//点样轴6X伺服控制
FB_SERVOAXIS_3(
	AXIS:= 点样轴6X ,                    //轴名称
	xEnable:=急停  ,                         //轴使能
	xStartupMotionAllowed:= FALSE, // startup axis ownership
	xHome:= 点样轴6XDATE.xHome,          //轴回零命令
	xJogPos:=点样轴6XDATE.xJogPos  ,     //轴正转命令
	xJogNeg:=点样轴6XDATE.xJogNeg  ,     //轴反转命令
	xStop:= 点样轴6XDATE.xStop ,         //轴停止命令
	xMoveAbs:= 点样轴6XDATE.xMoveAbs ,   //轴绝对定位命令
	xMoveRel:= 点样轴6XDATE.xMoveRel,    //轴相对定位命令
	XReset:= 点样轴6XDATE.XReset OR 复位 OR bSysReset,       //轴复位
	fAbsTarget:= 点样轴6XDATE.fAbsTarget ,  //轴绝对定位距离
	fRelTarget:=点样轴6XDATE.fRelTarget  ,  //轴相对移动距离
	fVelocity:= 点样轴6XDATE.fVelocity ,    //轴定位速度
	fAcc:=3500.0 ,              //轴加速度
	fDec:= 3500.0,              //轴减速度
	fJogVel:= 50.0 ,        //轴JOG速度
	bEnabled=> 点样轴6XDATE.bEnabled ,      //轴使能完成
	bHomed=> 回零完成6X ,          //轴回原点完成
	bBusy=> 点样轴6XDATE.bBusy ,            //轴运行中
	fActPos=>点样轴6XDATE.fActPos  ,        //轴当前位置
	fActVel=>点样轴6XDATE.fActVel  ,        //轴当前速度
	bAbMoveDone=>点样轴6XDATE.bAbMoveDone ,  //轴绝对定位完成
	bReMoveDone =>点样轴6XDATE.bReMoveDone ,);    //轴相对定位完成 
// startup alarm visibility axis 3
点样轴6XDATE.bError := FB_SERVOAXIS_3.bError AND NOT PLC_Startup_AlarmInhibit;
IF PLC_Startup_AlarmInhibit THEN
	点样轴6XDATE.iErrorCode := 0;
ELSE
	点样轴6XDATE.iErrorCode := FB_SERVOAXIS_3.iErrorCode;
END_IF
IF 回零完成6X THEN
	点样轴6XDATE.xHome := FALSE;
	点样轴6XDATE.bHomed := TRUE;
END_IF

//点样轴7Y伺服控制
FB_SERVOAXIS_4(
	AXIS:= 点样轴7Y ,                    //轴名称
	xEnable:=急停  ,                         //轴使能
	xStartupMotionAllowed:= FALSE, // startup axis ownership
	xHome:= 点样轴7YDATE.xHome,          //轴回零命令
	xJogPos:=点样轴7YDATE.xJogPos  ,     //轴正转命令
	xJogNeg:=点样轴7YDATE.xJogNeg  ,     //轴反转命令
	xStop:= 点样轴7YDATE.xStop ,         //轴停止命令
	xMoveAbs:= 点样轴7YDATE.xMoveAbs ,   //轴绝对定位命令
	xMoveRel:= 点样轴7YDATE.xMoveRel,    //轴相对定位命令
	XReset:= 点样轴7YDATE.XReset OR 复位 OR bSysReset,       //轴复位
	fAbsTarget:= 点样轴7YDATE.fAbsTarget ,  //轴绝对定位距离
	fRelTarget:=点样轴7YDATE.fRelTarget  ,  //轴相对移动距离
	fVelocity:= 点样轴7YDATE.fVelocity ,    //轴定位速度
	fAcc:=500.0 ,              //轴加速度
	fDec:= 500.0 ,              //轴减速度
	fJogVel:= 50.0 ,        //轴JOG速度
	bEnabled=> 点样轴7YDATE.bEnabled ,      //轴使能完成
	bHomed=>  回零完成7Y,          //轴回原点完成
	bBusy=> 点样轴7YDATE.bBusy ,            //轴运行中
	fActPos=>点样轴7YDATE.fActPos  ,        //轴当前位置
	fActVel=>点样轴7YDATE.fActVel  ,        //轴当前速度
	bAbMoveDone=>点样轴7YDATE.bAbMoveDone ,  //轴绝对定位完成
	bReMoveDone =>点样轴7YDATE.bReMoveDone ,);    //轴相对定位完成 
// startup alarm visibility axis 4
点样轴7YDATE.bError := FB_SERVOAXIS_4.bError AND NOT PLC_Startup_AlarmInhibit;
IF PLC_Startup_AlarmInhibit THEN
	点样轴7YDATE.iErrorCode := 0;
ELSE
	点样轴7YDATE.iErrorCode := FB_SERVOAXIS_4.iErrorCode;
END_IF
IF 回零完成7Y THEN
	点样轴7YDATE.xHome := FALSE;
	点样轴7YDATE.bHomed := TRUE;
END_IF

//拍照轴8Y伺服控制
FB_SERVOAXIS_5(
	AXIS:= 拍照轴8Y ,                    //轴名称
	xEnable:=急停  ,                         //轴使能
	xStartupMotionAllowed:= FALSE, // startup axis ownership
	xHome:= 拍照轴8YDATE.xHome,          //轴回零命令
	xJogPos:=拍照轴8YDATE.xJogPos  ,     //轴正转命令
	xJogNeg:=拍照轴8YDATE.xJogNeg  ,     //轴反转命令
	xStop:= 拍照轴8YDATE.xStop ,         //轴停止命令
	xMoveAbs:= 拍照轴8YDATE.xMoveAbs AND  刮板拍照遮光气缸上位 AND 刮板轴10ZDATE.fActPos<6 ,   //轴绝对定位命令
	xMoveRel:= 拍照轴8YDATE.xMoveRel,    //轴相对定位命令
	XReset:= 拍照轴8YDATE.XReset OR 复位 OR bSysReset,       //轴复位
	fAbsTarget:= 拍照轴8YDATE.fAbsTarget ,  //轴绝对定位距离
	fRelTarget:=拍照轴8YDATE.fRelTarget  ,  //轴相对移动距离
	fVelocity:= 拍照轴8YDATE.fVelocity ,    //轴定位速度
	fAcc:=500.0 ,              //轴加速度
	fDec:= 500.0 ,              //轴减速度
	fJogVel:= 50.0 ,        //轴JOG速度
	bEnabled=> 拍照轴8YDATE.bEnabled ,      //轴使能完成
	bHomed=> 回零完成8Y ,          //轴回原点完成
	bBusy=> 拍照轴8YDATE.bBusy ,            //轴运行中
	fActPos=>拍照轴8YDATE.fActPos  ,        //轴当前位置
	fActVel=>拍照轴8YDATE.fActVel  ,        //轴当前速度
	bAbMoveDone=>拍照轴8YDATE.bAbMoveDone ,  //轴绝对定位完成
	bReMoveDone =>拍照轴8YDATE.bReMoveDone ,);    //轴相对定位完成 
// startup alarm visibility axis 5
拍照轴8YDATE.bError := FB_SERVOAXIS_5.bError AND NOT PLC_Startup_AlarmInhibit;
IF PLC_Startup_AlarmInhibit THEN
	拍照轴8YDATE.iErrorCode := 0;
ELSE
	拍照轴8YDATE.iErrorCode := FB_SERVOAXIS_5.iErrorCode;
END_IF
	IF 回零完成8Y THEN
	拍照轴8YDATE.xHome := FALSE;
	拍照轴8YDATE.bHomed := TRUE;
END_IF

//刮板轴9X伺服控制
FB_SERVOAXIS_6(
	AXIS:= 刮板轴9X ,                    //轴名称
	xEnable:=急停  ,                         //轴使能
	xStartupMotionAllowed:= FALSE, // startup axis ownership
	xHome:= 刮板轴9XDATE.xHome,          //轴回零命令
	xJogPos:=刮板轴9XDATE.xJogPos  ,     //轴正转命令
	xJogNeg:=刮板轴9XDATE.xJogNeg  ,     //轴反转命令
	xStop:= 刮板轴9XDATE.xStop ,         //轴停止命令
	xMoveAbs:= 刮板轴9XDATE.xMoveAbs AND  刮板轴10ZDATE.fActPos<6,   //轴绝对定位命令
	xMoveRel:= 刮板轴9XDATE.xMoveRel,    //轴相对定位命令
	XReset:= 刮板轴9XDATE.XReset OR 复位 OR bSysReset,       //轴复位
	fAbsTarget:= 刮板轴9XDATE.fAbsTarget  ,  //轴绝对定位距离
	fRelTarget:=刮板轴9XDATE.fRelTarget  ,  //轴相对移动距离
	fVelocity:= 刮板轴9XDATE.fVelocity ,    //轴定位速度
	fAcc:=500.0 ,              //轴加速度
	fDec:= 500.0 ,              //轴减速度
	fJogVel:= 50.0 ,        //轴JOG速度
	bEnabled=> 刮板轴9XDATE.bEnabled ,      //轴使能完成
	bHomed=>  回零完成9X,          //轴回原点完成
	bBusy=> 刮板轴9XDATE.bBusy ,            //轴运行中
	fActPos=>刮板轴9XDATE.fActPos  ,        //轴当前位置
	fActVel=>刮板轴9XDATE.fActVel  ,        //轴当前速度
	bAbMoveDone=>刮板轴9XDATE.bAbMoveDone ,  //轴绝对定位完成
	bReMoveDone =>刮板轴9XDATE.bReMoveDone ,);    //轴相对定位完成 
// startup alarm visibility axis 6
刮板轴9XDATE.bError := FB_SERVOAXIS_6.bError AND NOT PLC_Startup_AlarmInhibit;
IF PLC_Startup_AlarmInhibit THEN
	刮板轴9XDATE.iErrorCode := 0;
ELSE
	刮板轴9XDATE.iErrorCode := FB_SERVOAXIS_6.iErrorCode;
END_IF
IF 回零完成9X THEN
	刮板轴9XDATE.xHome := FALSE;
	刮板轴9XDATE.bHomed := TRUE;
END_IF

//刮板轴10Z伺服控制
FB_SERVOAXIS_7(
	AXIS:= 刮板轴10Z ,                    //轴名称
	xEnable:=急停  ,                         //轴使能
	xStartupMotionAllowed:= FALSE, // startup axis ownership
	xHome:= 刮板轴10ZDATE.xHome,          //轴回零命令
	xJogPos:=刮板轴10ZDATE.xJogPos  ,     //轴正转命令
	xJogNeg:=刮板轴10ZDATE.xJogNeg  ,     //轴反转命令
	xStop:= 刮板轴10ZDATE.xStop ,         //轴停止命令
	xMoveAbs:= 刮板轴10ZDATE.xMoveAbs ,   //轴绝对定位命令
	xMoveRel:= 刮板轴10ZDATE.xMoveRel,    //轴相对定位命令
	XReset:= 刮板轴10ZDATE.XReset OR 复位 OR bSysReset,       //轴复位
	fAbsTarget:= 刮板轴10ZDATE.fAbsTarget ,  //轴绝对定位距离
	fRelTarget:=刮板轴10ZDATE.fRelTarget  ,  //轴相对移动距离
	fVelocity:= 刮板轴10ZDATE.fVelocity ,    //轴定位速度
	fAcc:=500.0  ,              //轴加速度
	fDec:= 500.0 ,              //轴减速度
	fJogVel:= 50.0 ,        //轴JOG速度
	bEnabled=> 刮板轴10ZDATE.bEnabled ,      //轴使能完成
	bHomed=> 回零完成10Z ,          //轴回原点完成
	bBusy=> 刮板轴10ZDATE.bBusy ,            //轴运行中
	fActPos=>刮板轴10ZDATE.fActPos  ,        //轴当前位置
	fActVel=>刮板轴10ZDATE.fActVel  ,        //轴当前速度
	bAbMoveDone=>刮板轴10ZDATE.bAbMoveDone ,  //轴绝对定位完成
	bReMoveDone =>刮板轴10ZDATE.bReMoveDone ,);    //轴相对定位完成 
// startup alarm visibility axis 7
刮板轴10ZDATE.bError := FB_SERVOAXIS_7.bError AND NOT PLC_Startup_AlarmInhibit;
IF PLC_Startup_AlarmInhibit THEN
	刮板轴10ZDATE.iErrorCode := 0;
ELSE
	刮板轴10ZDATE.iErrorCode := FB_SERVOAXIS_7.iErrorCode;
END_IF
IF 回零完成10Z THEN
	刮板轴10ZDATE.xHome := FALSE;
	刮板轴10ZDATE.bHomed := TRUE;
END_IF	
	
//地轨轴11Y伺服控制
FB_SERVOAXIS_8(
	AXIS:= 地轨轴11Y ,                    //轴名称
	xEnable:=急停  ,                         //轴使能
	xStartupMotionAllowed:= FALSE, // startup axis ownership
	xHome:= 地轨轴11YDATE.xHome,          //轴回零命令
	xJogPos:=地轨轴11YDATE.xJogPos  ,     //轴正转命令
	xJogNeg:=地轨轴11YDATE.xJogNeg  ,     //轴反转命令
	xStop:= 地轨轴11YDATE.xStop ,         //轴停止命令
	xMoveAbs:= 地轨轴11YDATE.xMoveAbs  ,   //轴绝对定位命令
	xMoveRel:= 地轨轴11YDATE.xMoveRel,    //轴相对定位命令
	XReset:= 地轨轴11YDATE.XReset OR 复位 OR bSysReset,       //轴复位
	fAbsTarget:= 地轨轴11YDATE.fAbsTarget ,  //轴绝对定位距离
	fRelTarget:=地轨轴11YDATE.fRelTarget  ,  //轴相对移动距离
	fVelocity:= 地轨轴11YDATE.fVelocity ,    //轴定位速度
	fAcc:=500.0 ,              //轴加速度
	fDec:= 500.0 ,              //轴减速度
	fJogVel:= 50.0 ,        //轴JOG速度
	bEnabled=> 地轨轴11YDATE.bEnabled ,      //轴使能完成
	bHomed=>  回零完成11Y,          //轴回原点完成
	bBusy=> 地轨轴11YDATE.bBusy ,            //轴运行中
	fActPos=>地轨轴11YDATE.fActPos  ,        //轴当前位置
	fActVel=>地轨轴11YDATE.fActVel  ,        //轴当前速度
	bAbMoveDone=>地轨轴11YDATE.bAbMoveDone ,  //轴绝对定位完成
	bReMoveDone =>地轨轴11YDATE.bReMoveDone ,);    //轴相对定位完成 
// startup alarm visibility axis 8
地轨轴11YDATE.bError := FB_SERVOAXIS_8.bError AND NOT PLC_Startup_AlarmInhibit;
IF PLC_Startup_AlarmInhibit THEN
	地轨轴11YDATE.iErrorCode := 0;
ELSE
	地轨轴11YDATE.iErrorCode := FB_SERVOAXIS_8.iErrorCode;
END_IF
IF 回零完成11Y THEN
	地轨轴11YDATE.xHome := FALSE;
	地轨轴11YDATE.bHomed := TRUE;
END_IF

//上样轴4X轴伺服控制
FB_SERVOAXIS_9(
	AXIS:= 上样轴4X轴 ,                    //轴名称
	xEnable:= 急停 AND NOT (Sampling_Servo_FreeMove AND (上样轴5Z轴DATE.fActPos < 3)) ,   //轴使能(去使能手推: 仅5Z抬起<3时放开4X)
	xStartupMotionAllowed:= ((PLC_Startup_State=50) OR (PLC_Startup_State=51)), // startup axis ownership
	xHome:= 上样轴4X轴DATE.xHome,          //轴回零命令
	xJogPos:=上样轴4X轴DATE.xJogPos  ,     //轴正转命令
	xJogNeg:=上样轴4X轴DATE.xJogNeg  ,     //轴反转命令
	xStop:= 上样轴4X轴DATE.xStop ,         //轴停止命令
	xMoveAbs:= 上样轴4X轴DATE.xMoveAbs AND  上样轴5Z轴DATE.fActPos<3 ,   //轴绝对定位命令
	xMoveRel:= 上样轴4X轴DATE.xMoveRel AND  上样轴5Z轴DATE.fActPos<3,    //轴相对定位命令
	XReset:= 上样轴4X轴DATE.XReset OR 复位 OR bSysReset,       //轴复位
	fAbsTarget:= 上样轴4X轴DATE.fAbsTarget ,  //轴绝对定位距离
	fRelTarget:=上样轴4X轴DATE.fRelTarget  ,  //轴相对移动距离
	fVelocity:= 上样轴4X轴DATE.fVelocity ,    //轴定位速度
	fAcc:=200.0 ,              //轴加速度
	fDec:= 200.0 ,              //轴减速度
	fJogVel:= 5.0,        //轴JOG速度
	bEnabled=> 上样轴4X轴DATE.bEnabled ,      //轴使能完成
	bHomed=>  回零完成4X,          //轴回原点完成
	bBusy=> 上样轴4X轴DATE.bBusy ,            //轴运行中
	fActPos=>上样轴4X轴DATE.fActPos  ,        //轴当前位置
	fActVel=>上样轴4X轴DATE.fActVel  ,        //轴当前速度
	bAbMoveDone=>上样轴4X轴DATE.bAbMoveDone ,  //轴绝对定位完成
	bReMoveDone =>上样轴4X轴DATE.bReMoveDone ,);    //轴相对定位完成 
// startup alarm visibility axis 9
上样轴4X轴DATE.bError := FB_SERVOAXIS_9.bError AND NOT PLC_Startup_AlarmInhibit;
IF PLC_Startup_AlarmInhibit THEN
	上样轴4X轴DATE.iErrorCode := 0;
ELSE
	上样轴4X轴DATE.iErrorCode := FB_SERVOAXIS_9.iErrorCode;
END_IF
IF 回零完成4X THEN
	上样轴4X轴DATE.xHome := FALSE;
	上样轴4X轴DATE.bHomed := TRUE;
END_IF
	%QB2216:= 27;             //回零模式27
IF NOT 急停 THEN
	上样轴4X轴DATE.bHomed := FALSE;
END_IF

//上样轴5Z轴伺服控制
FB_SERVOAXIS_10(
	AXIS:= 上样轴5Z轴 ,                    //轴名称
	xEnable:=急停  ,                         //轴使能
	xStartupMotionAllowed:= ((PLC_Startup_State=40) OR (PLC_Startup_State=41)), // startup axis ownership
	xHome:= 上样轴5Z轴DATE.xHome,          //轴回零命令
	xJogPos:=上样轴5Z轴DATE.xJogPos  ,     //轴正转命令
	xJogNeg:=上样轴5Z轴DATE.xJogNeg  ,     //轴反转命令
	xStop:= 上样轴5Z轴DATE.xStop ,         //轴停止命令
	xMoveAbs:= 上样轴5Z轴DATE.xMoveAbs ,   //轴绝对定位命令
	xMoveRel:= 上样轴5Z轴DATE.xMoveRel,    //轴相对定位命令
	XReset:= 上样轴5Z轴DATE.XReset OR 复位 OR bSysReset ,       //轴复位
	fAbsTarget:= 上样轴5Z轴DATE.fAbsTarget ,  //轴绝对定位距离
	fRelTarget:=上样轴5Z轴DATE.fRelTarget  ,  //轴相对移动距离
	fVelocity:= 上样轴5Z轴DATE.fVelocity ,    //轴定位速度
	fAcc:=300.0  ,              //轴加速度
	fDec:= 300.0 ,              //轴减速度
	fJogVel:= 20.0 ,        //轴JOG速度
	bEnabled=> 上样轴5Z轴DATE.bEnabled ,      //轴使能完成
	bHomed=> 回零完成5Z ,          //轴回原点完成
	bBusy=> 上样轴5Z轴DATE.bBusy ,            //轴运行中
	fActPos=>上样轴5Z轴DATE.fActPos  ,        //轴当前位置
	fActVel=>上样轴5Z轴DATE.fActVel  ,        //轴当前速度
	bAbMoveDone=>上样轴5Z轴DATE.bAbMoveDone ,   //轴绝对定位完成
	bReMoveDone =>上样轴5Z轴DATE.bReMoveDone , );   //轴相对定位完成 
// startup alarm visibility axis 10
上样轴5Z轴DATE.bError := FB_SERVOAXIS_10.bError AND NOT PLC_Startup_AlarmInhibit;
IF PLC_Startup_AlarmInhibit THEN
	上样轴5Z轴DATE.iErrorCode := 0;
ELSE
	上样轴5Z轴DATE.iErrorCode := FB_SERVOAXIS_10.iErrorCode;
END_IF
IF 回零完成5Z THEN
	上样轴5Z轴DATE.xHome := FALSE;
	上样轴5Z轴DATE.bHomed := TRUE;
END_IF
	%QB2228:= 27;                 //回零模式27
IF NOT 急停 THEN
	上样轴5Z轴DATE.bHomed := FALSE;
END_IF

//上样4X 与 打样3Y 实际使能镜像 -> 供上位机标定页显示真状态 (去使能手推时为 FALSE)
Sampling_Servo_Enabled := 上样轴4X轴DATE.bEnabled AND 打样瓶上料轴3YDATE.bEnabled;
END_ACTION

ACTION 位置示教:

//打样瓶上料轴3Y位置示教
FB_Teach_1(HMI_Servo:=HMI_打样瓶上料轴3Y , 
			Servo:=打样瓶上料轴3YDATE );
//点样轴6X位置示教
FB_Teach_2(HMI_Servo:=HMI_点样轴6X , 
			Servo:=点样轴6XDATE );
//点样轴7Y位置示教
FB_Teach_3(HMI_Servo:=HMI_点样轴7Y , 
			Servo:=点样轴7YDATE );			
//地轨轴11Y位置示教
FB_Teach_4(HMI_Servo:=HMI_地轨轴11Y , 
			Servo:=地轨轴11YDATE );			
//上样轴4X轴位置示教
FB_Teach_5(HMI_Servo:=HMI_上样轴4X轴 , 
			Servo:=上样轴4X轴DATE );			
//上样轴5Z轴位置示教
FB_Teach_6(HMI_Servo:=HMI_上样轴5Z轴 , 
			Servo:=上样轴5Z轴DATE );
END_ACTION

END_PROGRAM

// Device/Application/40_Man/initialization
PROGRAM initialization
VAR
	nTeachClear : INT;

END_VAR

玻璃上料轴1ZDATE.xHome := FALSE; 玻璃上料轴1ZDATE.xJogPos := FALSE; 玻璃上料轴1ZDATE.xJogNeg := FALSE;
玻璃上料轴1ZDATE.xMoveAbs := FALSE; 玻璃上料轴1ZDATE.xMoveRel := FALSE; 玻璃上料轴1ZDATE.xStop := FALSE; 玻璃上料轴1ZDATE.XReset := FALSE;
玻璃上料轴1ZDATE.bBusy := FALSE; 玻璃上料轴1ZDATE.bError := FALSE; 玻璃上料轴1ZDATE.iErrorCode := 0;
玻璃上料轴1ZDATE.bAbMoveDone := FALSE; 玻璃上料轴1ZDATE.bReMoveDone := FALSE;
玻璃上料轴2ZDATE.xHome := FALSE; 玻璃上料轴2ZDATE.xJogPos := FALSE; 玻璃上料轴2ZDATE.xJogNeg := FALSE;
玻璃上料轴2ZDATE.xMoveAbs := FALSE; 玻璃上料轴2ZDATE.xMoveRel := FALSE; 玻璃上料轴2ZDATE.xStop := FALSE; 玻璃上料轴2ZDATE.XReset := FALSE;
玻璃上料轴2ZDATE.bBusy := FALSE; 玻璃上料轴2ZDATE.bError := FALSE; 玻璃上料轴2ZDATE.iErrorCode := 0;
玻璃上料轴2ZDATE.bAbMoveDone := FALSE; 玻璃上料轴2ZDATE.bReMoveDone := FALSE;
打样瓶上料轴3YDATE.xHome := FALSE; 打样瓶上料轴3YDATE.xJogPos := FALSE; 打样瓶上料轴3YDATE.xJogNeg := FALSE;
打样瓶上料轴3YDATE.xMoveAbs := FALSE; 打样瓶上料轴3YDATE.xMoveRel := FALSE; 打样瓶上料轴3YDATE.xStop := FALSE; 打样瓶上料轴3YDATE.XReset := FALSE;
打样瓶上料轴3YDATE.bBusy := FALSE; 打样瓶上料轴3YDATE.bError := FALSE; 打样瓶上料轴3YDATE.iErrorCode := 0;
打样瓶上料轴3YDATE.bAbMoveDone := FALSE; 打样瓶上料轴3YDATE.bReMoveDone := FALSE;
点样轴6XDATE.xHome := FALSE; 点样轴6XDATE.xJogPos := FALSE; 点样轴6XDATE.xJogNeg := FALSE;
点样轴6XDATE.xMoveAbs := FALSE; 点样轴6XDATE.xMoveRel := FALSE; 点样轴6XDATE.xStop := FALSE; 点样轴6XDATE.XReset := FALSE;
点样轴6XDATE.bBusy := FALSE; 点样轴6XDATE.bError := FALSE; 点样轴6XDATE.iErrorCode := 0;
点样轴6XDATE.bAbMoveDone := FALSE; 点样轴6XDATE.bReMoveDone := FALSE;
点样轴7YDATE.xHome := FALSE; 点样轴7YDATE.xJogPos := FALSE; 点样轴7YDATE.xJogNeg := FALSE;
点样轴7YDATE.xMoveAbs := FALSE; 点样轴7YDATE.xMoveRel := FALSE; 点样轴7YDATE.xStop := FALSE; 点样轴7YDATE.XReset := FALSE;
点样轴7YDATE.bBusy := FALSE; 点样轴7YDATE.bError := FALSE; 点样轴7YDATE.iErrorCode := 0;
点样轴7YDATE.bAbMoveDone := FALSE; 点样轴7YDATE.bReMoveDone := FALSE;
拍照轴8YDATE.xHome := FALSE; 拍照轴8YDATE.xJogPos := FALSE; 拍照轴8YDATE.xJogNeg := FALSE;
拍照轴8YDATE.xMoveAbs := FALSE; 拍照轴8YDATE.xMoveRel := FALSE; 拍照轴8YDATE.xStop := FALSE; 拍照轴8YDATE.XReset := FALSE;
拍照轴8YDATE.bBusy := FALSE; 拍照轴8YDATE.bError := FALSE; 拍照轴8YDATE.iErrorCode := 0;
拍照轴8YDATE.bAbMoveDone := FALSE; 拍照轴8YDATE.bReMoveDone := FALSE;
刮板轴9XDATE.xHome := FALSE; 刮板轴9XDATE.xJogPos := FALSE; 刮板轴9XDATE.xJogNeg := FALSE;
刮板轴9XDATE.xMoveAbs := FALSE; 刮板轴9XDATE.xMoveRel := FALSE; 刮板轴9XDATE.xStop := FALSE; 刮板轴9XDATE.XReset := FALSE;
刮板轴9XDATE.bBusy := FALSE; 刮板轴9XDATE.bError := FALSE; 刮板轴9XDATE.iErrorCode := 0;
刮板轴9XDATE.bAbMoveDone := FALSE; 刮板轴9XDATE.bReMoveDone := FALSE;
刮板轴10ZDATE.xHome := FALSE; 刮板轴10ZDATE.xJogPos := FALSE; 刮板轴10ZDATE.xJogNeg := FALSE;
刮板轴10ZDATE.xMoveAbs := FALSE; 刮板轴10ZDATE.xMoveRel := FALSE; 刮板轴10ZDATE.xStop := FALSE; 刮板轴10ZDATE.XReset := FALSE;
刮板轴10ZDATE.bBusy := FALSE; 刮板轴10ZDATE.bError := FALSE; 刮板轴10ZDATE.iErrorCode := 0;
刮板轴10ZDATE.bAbMoveDone := FALSE; 刮板轴10ZDATE.bReMoveDone := FALSE;
地轨轴11YDATE.xHome := FALSE; 地轨轴11YDATE.xJogPos := FALSE; 地轨轴11YDATE.xJogNeg := FALSE;
地轨轴11YDATE.xMoveAbs := FALSE; 地轨轴11YDATE.xMoveRel := FALSE; 地轨轴11YDATE.xStop := FALSE; 地轨轴11YDATE.XReset := FALSE;
地轨轴11YDATE.bBusy := FALSE; 地轨轴11YDATE.bError := FALSE; 地轨轴11YDATE.iErrorCode := 0;
地轨轴11YDATE.bAbMoveDone := FALSE; 地轨轴11YDATE.bReMoveDone := FALSE;
上样轴4X轴DATE.xHome := FALSE; 上样轴4X轴DATE.xJogPos := FALSE; 上样轴4X轴DATE.xJogNeg := FALSE;
上样轴4X轴DATE.xMoveAbs := FALSE; 上样轴4X轴DATE.xMoveRel := FALSE; 上样轴4X轴DATE.xStop := FALSE; 上样轴4X轴DATE.XReset := FALSE;
上样轴4X轴DATE.bBusy := FALSE; 上样轴4X轴DATE.bError := FALSE; 上样轴4X轴DATE.iErrorCode := 0;
上样轴4X轴DATE.bAbMoveDone := FALSE; 上样轴4X轴DATE.bReMoveDone := FALSE;
上样轴5Z轴DATE.xHome := FALSE; 上样轴5Z轴DATE.xJogPos := FALSE; 上样轴5Z轴DATE.xJogNeg := FALSE;
上样轴5Z轴DATE.xMoveAbs := FALSE; 上样轴5Z轴DATE.xMoveRel := FALSE; 上样轴5Z轴DATE.xStop := FALSE; 上样轴5Z轴DATE.XReset := FALSE;
上样轴5Z轴DATE.bBusy := FALSE; 上样轴5Z轴DATE.bError := FALSE; 上样轴5Z轴DATE.iErrorCode := 0;
上样轴5Z轴DATE.bAbMoveDone := FALSE; 上样轴5Z轴DATE.bReMoveDone := FALSE;
	Z1JOG_pos := FALSE;
	Z1JOG_neg := FALSE;
	Z2JOG_POS := FALSE;
	Z2JOG_NEG := FALSE;
// Full download must invalidate retained teaching requests before normal motion can re-arm.
FOR nTeachClear:=1 TO 10 DO
	HMI_打样瓶上料轴3Y.execute[nTeachClear] := FALSE;
	HMI_打样瓶上料轴3Y.write[nTeachClear] := FALSE;
	HMI_点样轴6X.execute[nTeachClear] := FALSE;
	HMI_点样轴6X.write[nTeachClear] := FALSE;
	HMI_点样轴7Y.execute[nTeachClear] := FALSE;
	HMI_点样轴7Y.write[nTeachClear] := FALSE;
	HMI_地轨轴11Y.execute[nTeachClear] := FALSE;
	HMI_地轨轴11Y.write[nTeachClear] := FALSE;
	HMI_上样轴4X轴.execute[nTeachClear] := FALSE;
	HMI_上样轴4X轴.write[nTeachClear] := FALSE;
	HMI_上样轴5Z轴.execute[nTeachClear] := FALSE;
	HMI_上样轴5Z轴.write[nTeachClear] := FALSE;
END_FOR
一键回原点 := FALSE;
上样轴4X轴DATE.bHomed := FALSE;
上样轴5Z轴DATE.bHomed := FALSE;
HMI_HandWheel_3Y := FALSE; HMI_HandWheel_4X := FALSE; HMI_HandWheel_5Z := FALSE;
HMI_HandWheel_6X := FALSE; HMI_HandWheel_7Y := FALSE; HMI_HandWheel_8Y := FALSE;
HMI_HandWheel_9X := FALSE; HMI_HandWheel_10Z := FALSE; HMI_HandWheel_11Y := FALSE;
Sampling_Servo_FreeMove := FALSE;
PLC_Ready := FALSE;
PLC_Startup_AlarmInhibit := TRUE;
PLC_HandWheel_Active := FALSE;
PLC_Startup_State := 0;
PLC_Startup_ErrorCode := 0;
PLC_Deploy_CommitSeq := 0;
PLC_Deploy_Start := FALSE;
PLC_Deploy_Reset := FALSE;
PLC_Deploy_State := 0;
PLC_Deploy_ErrorCode := 0;
ECAT掉站报警 := FALSE;
伺服报警 := FALSE;
伺服未回原点报警 := FALSE;

END_PROGRAM

// Device/Application/25_FB_功能块/FB_Teach
FUNCTION_BLOCK FB_Teach
VAR_IN_OUT
	HMI_Servo: HMI_Servo;
	Servo: servo;
END_VAR
VAR
	i: INT;
END_VAR
VAR_INPUT
	Mode: INT;
	xEnble: BOOL;
END_VAR

IF Mode<>1 AND Servo.bEnabled AND SERVO.bHomed THEN    //没有在自动运行模式下，伺服使能
	//示教点位
	FOR i:=1 TO 10  DO
		IF HMI_Servo.write[i] THEN
		HMI_Servo.position[i]:=Servo.fActPos;
		END_IF
		//运动执行
		IF HMI_Servo.execute[i] THEN
			Servo.fAbsTarget:= HMI_Servo.position[i];
			Servo.xMoveAbs:=TRUE;
		END_IF
		//执行完毕复位
		IF Servo.bAbMoveDone OR Servo.bError  THEN
			Servo.xMoveAbs:=FALSE;
		END_IF
	END_FOR
	
END_IF

END_FUNCTION_BLOCK

// Device/Application/30_Ethercat任务/PLC_HandWheel_手轮
PROGRAM PLC_HandWheel_手轮
VAR
	FB_HandWheel_0: FB_HandWheel;
	HC_Counter_0: HC_Counter;
	bHandWheelAllowed: BOOL;
END_VAR

SMC_FreeEncoder.fActPosition := Encoder.fActPosition;

bHandWheelAllowed := 急停 AND (MODE_State<>1) AND NOT 手自动 AND PLC_Ready
	AND ((PLC_Deploy_State=0) OR (PLC_Deploy_State=30))
	AND PLC_Axis_CommOperational[3] AND PLC_Axis_CommOperational[4]
	AND PLC_Axis_CommOperational[5] AND PLC_Axis_CommOperational[6]
	AND PLC_Axis_CommOperational[7] AND PLC_Axis_CommOperational[8]
	AND PLC_Axis_CommOperational[9] AND PLC_Axis_CommOperational[10]
	AND PLC_Axis_CommOperational[11];

IF NOT bHandWheelAllowed THEN
	HMI_HandWheel_3Y := FALSE; HMI_HandWheel_4X := FALSE; HMI_HandWheel_5Z := FALSE;
	HMI_HandWheel_6X := FALSE; HMI_HandWheel_7Y := FALSE; HMI_HandWheel_8Y := FALSE;
	HMI_HandWheel_9X := FALSE; HMI_HandWheel_10Z := FALSE; HMI_HandWheel_11Y := FALSE;
END_IF

HC_Counter_0(Axis := Encoder, Enable := bHandWheelAllowed);
FB_HandWheel_0(
	Axis_Spindle := SMC_FreeEncoder,
	AXIS_1 := 打样瓶上料轴3Y,
	AXIS_2 := 上样轴4X轴,
	AXIS_3 := 上样轴5Z轴,
	AXIS_4 := 点样轴6X,
	AXIS_5 := 点样轴7Y,
	AXIS_6 := 拍照轴8Y,
	AXIS_7 := 刮板轴9X,
	AXIS_8 := 刮板轴10Z,
	AXIS_9 := 地轨轴11Y,
	Enable := bHandWheelAllowed,
	Speed_X1 := 倍率X1,
	Speed_X10 := 倍率X10,
	Speed_X100 := 倍率X100,
	Reset := 复位,
	HandWheel_3Y := HMI_HandWheel_3Y,
	HandWheel_4X := HMI_HandWheel_4X,
	HandWheel_5Z := HMI_HandWheel_5Z,
	HandWheel_6X := HMI_HandWheel_6X,
	HandWheel_7Y := HMI_HandWheel_7Y,
	HandWheel_8Y := HMI_HandWheel_8Y,
	HandWheel_9X := HMI_HandWheel_9X,
	HandWheel_10Z := HMI_HandWheel_10Z,
	HandWheel_11Y := HMI_HandWheel_11Y,
	xStop_1 => 打样瓶上料轴3YDATE.xStop,
	xStop_2 => 上样轴4X轴DATE.xStop,
	xStop_3 => 上样轴5Z轴DATE.xStop,
	xStop_4 => 点样轴6XDATE.xStop,
	xStop_5 => 点样轴7YDATE.xStop,
	xStop_6 => 拍照轴8YDATE.xStop,
	xStop_7 => 刮板轴9XDATE.xStop,
	xStop_8 => 刮板轴10ZDATE.xStop,
	xStop_9 => 地轨轴11YDATE.xStop);
PLC_HandWheel_Active := FB_HandWheel_0.Active;

END_PROGRAM

// Device/Application/25_FB_功能块/FB_HandWheel
FUNCTION_BLOCK FB_HandWheel
VAR_IN_OUT
	Axis_Spindle: AXIS_REF_SM3;
	AXIS_1: AXIS_REF_SM3;
	AXIS_2: AXIS_REF_SM3;
	AXIS_3: AXIS_REF_SM3;
	AXIS_4: AXIS_REF_SM3;
	AXIS_5: AXIS_REF_SM3;
	AXIS_6: AXIS_REF_SM3;
	AXIS_7: AXIS_REF_SM3;
	AXIS_8: AXIS_REF_SM3;
	AXIS_9: AXIS_REF_SM3;
END_VAR
VAR_INPUT
	Enable: BOOL;
	Speed_X1: BOOL;
	Speed_X10: BOOL;
	Speed_X100: BOOL;
	Reset: BOOL;
	HandWheel_3Y: BOOL;
	HandWheel_4X: BOOL;
	HandWheel_5Z: BOOL;
	HandWheel_6X: BOOL;
	HandWheel_7Y: BOOL;
	HandWheel_8Y: BOOL;
	HandWheel_9X: BOOL;
	HandWheel_10Z: BOOL;
	HandWheel_11Y: BOOL;
END_VAR
VAR_OUTPUT
	xStop_1: BOOL;
	xStop_2: BOOL;
	xStop_3: BOOL;
	xStop_4: BOOL;
	xStop_5: BOOL;
	xStop_6: BOOL;
	xStop_7: BOOL;
	xStop_8: BOOL;
	xStop_9: BOOL;
	Active: BOOL;
	Error: BOOL;
	ErrorID: WORD;
END_VAR
VAR
	MC_GearIn_1: MC_GearIn;
	MC_GearIn_2: MC_GearIn;
	MC_GearIn_3: MC_GearIn;
	MC_GearIn_4: MC_GearIn;
	MC_GearIn_5: MC_GearIn;
	MC_GearIn_6: MC_GearIn;
	MC_GearIn_7: MC_GearIn;
	MC_GearIn_8: MC_GearIn;
	MC_GearIn_9: MC_GearIn;
	MC_GearOut_1: MC_GearOut;
	MC_GearOut_2: MC_GearOut;
	MC_GearOut_3: MC_GearOut;
	MC_GearOut_4: MC_GearOut;
	MC_GearOut_5: MC_GearOut;
	MC_GearOut_6: MC_GearOut;
	MC_GearOut_7: MC_GearOut;
	MC_GearOut_8: MC_GearOut;
	MC_GearOut_9: MC_GearOut;
	R_TRIG_1: R_TRIG;
	R_TRIG_2: R_TRIG;
	R_TRIG_3: R_TRIG;
	R_TRIG_5: R_TRIG;
	R_TRIG_6: R_TRIG;
	R_TRIG_7: R_TRIG;
	R_TRIG_8: R_TRIG;
	R_TRIG_9: R_TRIG;
	R_TRIG_10: R_TRIG;
	R_TRIG_11: R_TRIG;
	R_TRIG_12: R_TRIG;
	R_TRIG_13: R_TRIG;
	F_TRIG_1: F_TRIG;
	F_TRIG_2: F_TRIG;
	F_TRIG_3: F_TRIG;
	F_TRIG_4: F_TRIG;
	F_TRIG_5: F_TRIG;
	F_TRIG_6: F_TRIG;
	F_TRIG_7: F_TRIG;
	F_TRIG_8: F_TRIG;
	F_TRIG_9: F_TRIG;
	iDenominator: UDINT := 100;
	iMolecule: INT := 1;
END_VAR

// Every PLCopen gearing FB is called cyclically. Dropping Enable forces GearOut.
IF Speed_X1 THEN
	iDenominator := 100;
ELSIF Speed_X10 THEN
	iDenominator := 10;
ELSIF Speed_X100 THEN
	iDenominator := 1;
END_IF
R_TRIG_1(CLK := Enable AND Speed_X1);
R_TRIG_2(CLK := Enable AND Speed_X10);
R_TRIG_3(CLK := Enable AND Speed_X100);

R_TRIG_5(CLK := Enable AND HandWheel_3Y);
F_TRIG_1(CLK := Enable AND HandWheel_3Y);
MC_GearIn_1(
	Master := Axis_Spindle,
	Slave := AXIS_1,
	Execute := Enable AND (R_TRIG_5.Q
		OR ((R_TRIG_1.Q OR R_TRIG_2.Q OR R_TRIG_3.Q) AND HandWheel_3Y)),
	RatioNumerator := iMolecule,
	RatioDenominator := iDenominator,
	Acceleration := 500,
	Deceleration := 800);
MC_GearOut_1(
	Slave := AXIS_1,
	Execute := (F_TRIG_1.Q OR NOT Enable) AND MC_GearIn_1.InGear,
	Done => xStop_1);

R_TRIG_6(CLK := Enable AND HandWheel_4X);
F_TRIG_2(CLK := Enable AND HandWheel_4X);
MC_GearIn_2(
	Master := Axis_Spindle,
	Slave := AXIS_2,
	Execute := Enable AND (R_TRIG_6.Q
		OR ((R_TRIG_1.Q OR R_TRIG_2.Q OR R_TRIG_3.Q) AND HandWheel_4X)),
	RatioNumerator := iMolecule,
	RatioDenominator := iDenominator,
	Acceleration := 500,
	Deceleration := 800);
MC_GearOut_2(
	Slave := AXIS_2,
	Execute := (F_TRIG_2.Q OR NOT Enable) AND MC_GearIn_2.InGear,
	Done => xStop_2);

R_TRIG_7(CLK := Enable AND HandWheel_5Z);
F_TRIG_3(CLK := Enable AND HandWheel_5Z);
MC_GearIn_3(
	Master := Axis_Spindle,
	Slave := AXIS_3,
	Execute := Enable AND (R_TRIG_7.Q
		OR ((R_TRIG_1.Q OR R_TRIG_2.Q OR R_TRIG_3.Q) AND HandWheel_5Z)),
	RatioNumerator := iMolecule,
	RatioDenominator := iDenominator,
	Acceleration := 500,
	Deceleration := 800);
MC_GearOut_3(
	Slave := AXIS_3,
	Execute := (F_TRIG_3.Q OR NOT Enable) AND MC_GearIn_3.InGear,
	Done => xStop_3);

R_TRIG_8(CLK := Enable AND HandWheel_6X);
F_TRIG_4(CLK := Enable AND HandWheel_6X);
MC_GearIn_4(
	Master := Axis_Spindle,
	Slave := AXIS_4,
	Execute := Enable AND (R_TRIG_8.Q
		OR ((R_TRIG_1.Q OR R_TRIG_2.Q OR R_TRIG_3.Q) AND HandWheel_6X)),
	RatioNumerator := iMolecule,
	RatioDenominator := iDenominator,
	Acceleration := 500,
	Deceleration := 800);
MC_GearOut_4(
	Slave := AXIS_4,
	Execute := (F_TRIG_4.Q OR NOT Enable) AND MC_GearIn_4.InGear,
	Done => xStop_4);

R_TRIG_9(CLK := Enable AND HandWheel_7Y);
F_TRIG_5(CLK := Enable AND HandWheel_7Y);
MC_GearIn_5(
	Master := Axis_Spindle,
	Slave := AXIS_5,
	Execute := Enable AND (R_TRIG_9.Q
		OR ((R_TRIG_1.Q OR R_TRIG_2.Q OR R_TRIG_3.Q) AND HandWheel_7Y)),
	RatioNumerator := iMolecule,
	RatioDenominator := iDenominator,
	Acceleration := 500,
	Deceleration := 800);
MC_GearOut_5(
	Slave := AXIS_5,
	Execute := (F_TRIG_5.Q OR NOT Enable) AND MC_GearIn_5.InGear,
	Done => xStop_5);

R_TRIG_10(CLK := Enable AND HandWheel_8Y);
F_TRIG_6(CLK := Enable AND HandWheel_8Y);
MC_GearIn_6(
	Master := Axis_Spindle,
	Slave := AXIS_6,
	Execute := Enable AND (R_TRIG_10.Q
		OR ((R_TRIG_1.Q OR R_TRIG_2.Q OR R_TRIG_3.Q) AND HandWheel_8Y)),
	RatioNumerator := iMolecule,
	RatioDenominator := iDenominator,
	Acceleration := 500,
	Deceleration := 800);
MC_GearOut_6(
	Slave := AXIS_6,
	Execute := (F_TRIG_6.Q OR NOT Enable) AND MC_GearIn_6.InGear,
	Done => xStop_6);

R_TRIG_11(CLK := Enable AND HandWheel_9X);
F_TRIG_7(CLK := Enable AND HandWheel_9X);
MC_GearIn_7(
	Master := Axis_Spindle,
	Slave := AXIS_7,
	Execute := Enable AND (R_TRIG_11.Q
		OR ((R_TRIG_1.Q OR R_TRIG_2.Q OR R_TRIG_3.Q) AND HandWheel_9X)),
	RatioNumerator := iMolecule,
	RatioDenominator := iDenominator,
	Acceleration := 500,
	Deceleration := 800);
MC_GearOut_7(
	Slave := AXIS_7,
	Execute := (F_TRIG_7.Q OR NOT Enable) AND MC_GearIn_7.InGear,
	Done => xStop_7);

R_TRIG_12(CLK := Enable AND HandWheel_10Z);
F_TRIG_8(CLK := Enable AND HandWheel_10Z);
MC_GearIn_8(
	Master := Axis_Spindle,
	Slave := AXIS_8,
	Execute := Enable AND (R_TRIG_12.Q
		OR ((R_TRIG_1.Q OR R_TRIG_2.Q OR R_TRIG_3.Q) AND HandWheel_10Z)),
	RatioNumerator := iMolecule,
	RatioDenominator := iDenominator,
	Acceleration := 500,
	Deceleration := 800);
MC_GearOut_8(
	Slave := AXIS_8,
	Execute := (F_TRIG_8.Q OR NOT Enable) AND MC_GearIn_8.InGear,
	Done => xStop_8);

R_TRIG_13(CLK := Enable AND HandWheel_11Y);
F_TRIG_9(CLK := Enable AND HandWheel_11Y);
MC_GearIn_9(
	Master := Axis_Spindle,
	Slave := AXIS_9,
	Execute := Enable AND (R_TRIG_13.Q
		OR ((R_TRIG_1.Q OR R_TRIG_2.Q OR R_TRIG_3.Q) AND HandWheel_11Y)),
	RatioNumerator := iMolecule,
	RatioDenominator := iDenominator,
	Acceleration := 500,
	Deceleration := 800);
MC_GearOut_9(
	Slave := AXIS_9,
	Execute := (F_TRIG_9.Q OR NOT Enable) AND MC_GearIn_9.InGear,
	Done => xStop_9);

Active := MC_GearIn_1.InGear OR MC_GearIn_1.Busy OR MC_GearOut_1.Busy OR MC_GearIn_2.InGear OR MC_GearIn_2.Busy OR MC_GearOut_2.Busy OR MC_GearIn_3.InGear OR MC_GearIn_3.Busy OR MC_GearOut_3.Busy OR MC_GearIn_4.InGear OR MC_GearIn_4.Busy OR MC_GearOut_4.Busy OR MC_GearIn_5.InGear OR MC_GearIn_5.Busy OR MC_GearOut_5.Busy OR MC_GearIn_6.InGear OR MC_GearIn_6.Busy OR MC_GearOut_6.Busy OR MC_GearIn_7.InGear OR MC_GearIn_7.Busy OR MC_GearOut_7.Busy OR MC_GearIn_8.InGear OR MC_GearIn_8.Busy OR MC_GearOut_8.Busy OR MC_GearIn_9.InGear OR MC_GearIn_9.Busy OR MC_GearOut_9.Busy;
Error := MC_GearIn_1.Error OR MC_GearOut_1.Error OR MC_GearIn_2.Error OR MC_GearOut_2.Error OR MC_GearIn_3.Error OR MC_GearOut_3.Error OR MC_GearIn_4.Error OR MC_GearOut_4.Error OR MC_GearIn_5.Error OR MC_GearOut_5.Error OR MC_GearIn_6.Error OR MC_GearOut_6.Error OR MC_GearIn_7.Error OR MC_GearOut_7.Error OR MC_GearIn_8.Error OR MC_GearOut_8.Error OR MC_GearIn_9.Error OR MC_GearOut_9.Error;
ErrorID := 0;
IF MC_GearIn_1.Error THEN ErrorID := MC_GearIn_1.ErrorID;
ELSIF MC_GearOut_1.Error THEN ErrorID := MC_GearOut_1.ErrorID;
ELSIF MC_GearIn_2.Error THEN ErrorID := MC_GearIn_2.ErrorID;
ELSIF MC_GearOut_2.Error THEN ErrorID := MC_GearOut_2.ErrorID;
ELSIF MC_GearIn_3.Error THEN ErrorID := MC_GearIn_3.ErrorID;
ELSIF MC_GearOut_3.Error THEN ErrorID := MC_GearOut_3.ErrorID;
ELSIF MC_GearIn_4.Error THEN ErrorID := MC_GearIn_4.ErrorID;
ELSIF MC_GearOut_4.Error THEN ErrorID := MC_GearOut_4.ErrorID;
ELSIF MC_GearIn_5.Error THEN ErrorID := MC_GearIn_5.ErrorID;
ELSIF MC_GearOut_5.Error THEN ErrorID := MC_GearOut_5.ErrorID;
ELSIF MC_GearIn_6.Error THEN ErrorID := MC_GearIn_6.ErrorID;
ELSIF MC_GearOut_6.Error THEN ErrorID := MC_GearOut_6.ErrorID;
ELSIF MC_GearIn_7.Error THEN ErrorID := MC_GearIn_7.ErrorID;
ELSIF MC_GearOut_7.Error THEN ErrorID := MC_GearOut_7.ErrorID;
ELSIF MC_GearIn_8.Error THEN ErrorID := MC_GearIn_8.ErrorID;
ELSIF MC_GearOut_8.Error THEN ErrorID := MC_GearOut_8.ErrorID;
ELSIF MC_GearIn_9.Error THEN ErrorID := MC_GearIn_9.ErrorID;
ELSIF MC_GearOut_9.Error THEN ErrorID := MC_GearOut_9.ErrorID;
END_IF

END_FUNCTION_BLOCK

// Device/Application/40_Man/Expand_process_展开流程
PROGRAM Expand_process_展开流程
VAR
	清洗STEP: INT;
	TON_0: TON;
	润洗展缸STEP: INT;
	TON_1: TON;
	TON_2: TON;
	上液step: INT;
	放硅胶板step: INT;
	展开step: INT;
	TON_3: TON;
	TON_4: TON;
	stepTimer   : TON;       // 步骤内通用定时器
    targetTank  : INT;       // 本轮 prep 的目标缸号（锁存值）
    targetGroup : INT;       // 推导的组号（1 或 2）
    targetNum   : INT;       // 推导的组内序号（1-4）
    i           : INT;       // 循环索引
	ton3s: TON;
	初始化step: INT;
	泵初始化完成: BOOL;
	R_TRIG: ARRAY[1..10] OF R_TRIG;
	TON: ARRAY[1..10] OF TON;
	润洗计数: INT;
	上液计数: INT;
	L2_StartTrig : R_TRIG;            // Develop_L2_Start 上升沿检测器
END_VAR

IF (Develop_ControlMode = 1) AND (Develop_L2_State = 10) THEN
	IF (NOT 急停) OR (MODE_State <> 1) THEN
		Develop_L2_ErrorCode    := 401;
		Develop_L2_SafeState    := 90;
		Develop_L2_Retryable    := FALSE;
		Develop_L2_CompletedSeq := Develop_L2_AcceptedSeq;
		Develop_L2_State        := 50;     // INTERRUPTED
	END_IF
END_IF

IF 大真空泵站位[0] OR 大真空泵站位[1] OR 大真空泵站位[2] OR 大真空泵站位[3] OR 大真空泵站位[4] OR 大真空泵站位[5] OR 大真空泵站位[6] OR 大真空泵站位[7] OR 大真空泵站位[8] OR 大真空泵站位[9] OR 大真空泵站位[10] OR 大真空泵站位[11] THEN
	大真空泵自动:=TRUE;
	ELSE
	大真空泵自动:=FALSE;
END_IF

// ── 1. 急停联锁（最高优先级）──
IF NOT 急停 THEN
    Expand_Step  := 0;
    Expand_Done  := FALSE;
    Expand_Error := TRUE;
    Expand_Busy  := FALSE;
	大真空泵站位[1]:=FALSE;
	大真空泵站位[2]:=FALSE;
	大真空泵站位[3]:=FALSE;
	大真空泵站位[4]:=FALSE;
	大真空泵站位[5]:=FALSE;
	大真空泵站位[6]:=FALSE;
	大真空泵站位[7]:=FALSE;
	大真空泵站位[8]:=FALSE;
	清洗STEP:=0;
	润洗展缸STEP:=0;
	上液step:=0;
	放硅胶板step:=0;
	展开step:=0;
	初始化step:=0;
	泵初始化完成:=FALSE;
	润洗计数:=0;
	上液计数:=0;
    // 急停时将所有 Prepping 状态的缸标记为 Error
    FOR i := 1 TO 8 DO
        IF Tank_State[i] = 10 THEN
            Tank_State[i] := 90;
        END_IF
    END_FOR
    stepTimer(IN := FALSE, PT := T#0S);
    RETURN;
END_IF

// ── 2. 复位脉冲（用于错误恢复 / 强制清状态）──
IF Expand_Reset THEN
    // 清序列器自身状态
    Expand_Step  := 0;
    Expand_Done  := FALSE;
    Expand_Error := FALSE;
    Expand_Busy  := FALSE;
    stepTimer(IN := FALSE, PT := T#0S);
    // 若有活跃 prep 目标缸，将其标记为 Error（避免孤儿缸）
    IF targetTank >= 1 AND targetTank <= 8 THEN
        IF Tank_State[targetTank] = 10 THEN
            Tank_State[targetTank] := 90;
        END_IF
    END_IF
    // 注：Tank_State[90] 的缸由 PC 写 0 复位（ResourceManager.release()）
    RETURN;
END_IF

// ── 3. Enable=FALSE 时清 Done（次周期复位握手）──
IF NOT Expand_Enable THEN
    Expand_Done := FALSE;
END_IF


// ── 4. 派生 Expand_Busy（写者唯一：本 POU 是唯一写者，禁止他处赋值）──
Expand_Busy := (Expand_Step >= 10)
              AND (Expand_Step <= 80)
              AND (NOT Expand_Done);

IF MODE_State=1 THEN	
	IF Develop_ControlMode = 0 THEN       // LEGACY (默认)
		CASE Expand_Step OF
			0:  // ═══ 空闲：等待 Enable 上升 ═══
				IF Expand_Enable AND (NOT Expand_Done) THEN
					// 读取目标缸号并校验
					targetTank := Expand_Target_Tank;
		
					// 校验：目标缸号必须在 1-8 范围内
					IF targetTank < 1 OR targetTank > 8 THEN
						Expand_Error := TRUE;
						Expand_Step := 90;
					// 校验：目标缸必须处于 Idle 状态（防止重复 prep）
					ELSIF Tank_State[targetTank] <> 0 THEN
						Expand_Error := TRUE;
						Expand_Step := 90;
					ELSE
						// 自动推导 Group 和 Number
						targetGroup := (targetTank - 1) / 4 + 1;   // 1-4→Group1, 5-8→Group2
						targetNum   := (targetTank - 1) MOD 4 + 1; // 组内序号 1-4
		
						// 写入协议变量（供 FB 调用使用）
						Expand_Group  := targetGroup;
						Expand_Number := targetNum;
		
						// 标记目标缸进入 Prepping 状态
						Tank_State[targetTank] := 10;
		
						// 推进到 Step 10
						Expand_Step := 5;
						stepTimer(IN := FALSE, PT := T#0S);  // 复位定时器
					END_IF
				END_IF
			 5:                //初始化
				
					A00_initialization_初始化();
					IF  泵初始化完成 THEN
						
						泵初始化完成:=FALSE;
						Expand_Step:=10;
					END_IF
			10: // ═══ 润洗/清洗（Expand_Mode_Flag=0→缸模式；=1→管路模式）═══
				// 润洗/清洗操作针对 targetTank 对应的泵组
				IF Expand_Mode_Flag=0  THEN
					A20_clean_expand_润洗展缸();
				ELSIF Expand_Mode_Flag=1 THEN
					A10_pipeline_cleaning_清洗管路();
				END_IF
				IF Expand_Group_clean_OK THEN
					Expand_Group_clean_OK:=FALSE;
					Expand_Step:=20;
				END_IF
			 20: // ═══ 上液（展开剂加入目标展缸）═══
				IF Expand_Group>0 AND Expand_Number>0 THEN
					A40_up_liquid_上液();
				END_IF
				IF Expand_up_liquid_OK THEN
					Expand_up_liquid_OK:=FALSE;
					Expand_Step:=30;
				END_IF
			30: // ═══ 放硅胶板（机械臂+传感器自治）═══
				A30_silica_gel_plate_放硅胶板();
				IF Expand_silica_gel_plate_OK THEN
					Expand_silica_gel_plate_OK:=FALSE;
					Expand_Step:=40;
				END_IF
		
			40: // ═══ 【关键变更】交付至展开态 —— 立即释放序列器 ═══
				Tank_State[targetTank] := 40;
		
				// 标记 prep 完成，释放序列器
				Expand_Done := TRUE;
				Expand_Busy := FALSE;
				Expand_Step := 0;
		
				// 序列器已归零，可接受下一个 prep 请求
				// 实际展开由缸自身"静置"完成，排液由独立子程序 PRG_TankDrain 处理
		
			90: // ═══ 故障态：等待外部 Expand_Reset 脉冲 ═══
				Expand_Error := TRUE;   // 故障态本身不动作，仅等待顶部复位逻辑
				
		END_CASE
	ELSE
		(* L2 派发已由 PLC_MainPRG 每扫描调用的 50_action/Develop_L2 承担;
		   旧 Develop_L2_Dispatch 码表过期 (30/40) 且 code50 卡 Tank_State=40 前置,
		   若在此启用会与活派发器双写 Develop_L2_* 通道, 故拆除.
		   spec: docs/superpowers/specs/2026-07-14-develop-drain-l2-migration-design.md *)
	END_IF
END_IF

ACTION Develop_L2_Dispatch:
// 功能:
//   展开 L2 统一动作通道派发器。仅在 MODE_State=1 且 Develop_ControlMode=1 时由
//   POU body 调用 (与 legacy CASE Expand_Step 互斥, 单写者)。接受动作时由
//   Expand_Target_Tank 派生 Expand_Group/Expand_Number, 再路由到对应 A 动作;
//   drain 桥接 Tank_Drain 数组。
// 参数: 无 (Expand_Target_Tank 经全局传入)。返回: 无 (经 Develop_L2_* 反馈)。
L2_StartTrig(CLK := Develop_L2_Start);

CASE Develop_L2_State OF

	0:  // ═══ IDLE ═══
		Develop_L2_Step := 0;
		IF L2_StartTrig.Q THEN
			Develop_L2_AcceptedSeq := Develop_L2_RequestSeq;
			Develop_L2_ActiveCode  := Develop_L2_ActionCode;
			Develop_L2_ErrorCode   := 0;
			Develop_L2_Retryable   := FALSE;
			// 所有 Develop 动作都需要目标缸号确定泵组, 先校验并派生
			targetTank := Expand_Target_Tank;
			IF (targetTank < 1) OR (targetTank > 8) THEN
				Develop_L2_ErrorCode    := 102;        // 缸号超范围
				Develop_L2_Retryable    := TRUE;
				Develop_L2_CompletedSeq := Develop_L2_AcceptedSeq;
				Develop_L2_State        := 30;         // REJECTED
			ELSIF (Develop_L2_ActionCode = 10) OR (Develop_L2_ActionCode = 20)
			      OR (Develop_L2_ActionCode = 30) OR (Develop_L2_ActionCode = 40) THEN
				// 派生泵组 (复用 legacy step 0 公式)
				targetGroup := (targetTank - 1) / 4 + 1;
				targetNum   := (targetTank - 1) MOD 4 + 1;
				Expand_Group  := targetGroup;
				Expand_Number := targetNum;
				// 复位 A 动作局部步进 (镜像本 POU 急停复位集合)
				清洗STEP := 0;
				润洗展缸STEP := 0;
				上液step := 0;
				初始化step := 0;
				泵初始化完成 := FALSE;
				润洗计数 := 0;
				上液计数 := 0;
				Develop_L2_SafeState := 0;
				Develop_L2_State := 10;                // RUNNING
			ELSIF Develop_L2_ActionCode = 50 THEN
				// drain: 前置缸必须处于 Developing(40)
				IF Tank_State[targetTank] = 40 THEN
					Tank_Drain_Enable[targetTank] := TRUE;
					Develop_L2_State := 10;            // RUNNING
				ELSE
					Develop_L2_ErrorCode    := 501;    // 缸非 Developing, 不可排液
					Develop_L2_Retryable    := TRUE;
					Develop_L2_CompletedSeq := Develop_L2_AcceptedSeq;
					Develop_L2_State        := 30;     // REJECTED
				END_IF
			ELSE
				Develop_L2_ErrorCode    := 101;        // 未知动作码
				Develop_L2_Retryable    := TRUE;
				Develop_L2_CompletedSeq := Develop_L2_AcceptedSeq;
				Develop_L2_State        := 30;         // REJECTED
			END_IF
		END_IF

	10: // ═══ RUNNING ═══
		CASE Develop_L2_ActiveCode OF
			10:  // 初始化 (目标泵组)
				A00_initialization_初始化();
				Develop_L2_Step := 初始化step;
				IF 泵初始化完成 THEN
					泵初始化完成 := FALSE;
					Develop_L2_SafeState    := 10;   // READY
					Develop_L2_CompletedSeq := Develop_L2_AcceptedSeq;
					Develop_L2_State        := 20;   // DONE
				END_IF
			20:  // 清洗管路
				A10_pipeline_cleaning_清洗管路();
				Develop_L2_Step := 清洗STEP;
				IF Expand_Group_clean_OK THEN
					Expand_Group_clean_OK := FALSE;
					Develop_L2_CompletedSeq := Develop_L2_AcceptedSeq;
					Develop_L2_State        := 20;   // DONE
				END_IF
			30:  // 润洗展缸 (目标缸)
				A20_clean_expand_润洗展缸();
				Develop_L2_Step := 润洗展缸STEP;
				IF Expand_Group_clean_OK THEN
					Expand_Group_clean_OK := FALSE;
					Develop_L2_CompletedSeq := Develop_L2_AcceptedSeq;
					Develop_L2_State        := 20;   // DONE
				END_IF
			40:  // 上液 (目标缸)
				IF (Expand_Group > 0) AND (Expand_Number > 0) THEN
					A40_up_liquid_上液();
				END_IF
				Develop_L2_Step := 上液step;
				IF Expand_up_liquid_OK THEN
					Expand_up_liquid_OK := FALSE;
					Develop_L2_CompletedSeq := Develop_L2_AcceptedSeq;
					Develop_L2_State        := 20;   // DONE
				END_IF
			50:  // 排液 (桥接 Tank_Drain 数组; A50/PRG_TankDrain 独立并行推进)
				Develop_L2_Step := Tank_State[targetTank];
				IF Tank_Drain_Done[targetTank] THEN
					Develop_L2_SafeState    := 10;   // READY (缸已排空待取板)
					Develop_L2_CompletedSeq := Develop_L2_AcceptedSeq;
					Develop_L2_State        := 20;   // DONE
				END_IF
		END_CASE

	20, 30, 40, 50:  // ═══ 终态 ═══
		IF (NOT Develop_L2_Start) OR Develop_L2_Reset THEN
			// drain 完成后回 IDLE 时撤除 Enable (Tank_State 由上位机写 0 释放)
			IF Develop_L2_ActiveCode = 50 THEN
				Tank_Drain_Enable[targetTank] := FALSE;
			END_IF
			Develop_L2_State := 0;
		END_IF

END_CASE
END_ACTION

ACTION A00_initialization_初始化:
R_TRIG[1](CLK:=%MX2005.5 , Q=> );  //泵空闲中
R_TRIG[2](CLK:=%MX2005.5 , Q=> );  //泵空闲中

CASE 初始化step OF
	0:
		润洗展缸STEP:=0;
		清洗STEP:=0;
		上液step:=0;
		放硅胶板step:=0;
		展开step:=0;
		expand_initialization_OK:=FALSE;
		Expand_Group_clean_OK:=FALSE;
		Expand_up_liquid_OK:=FALSE;
		Expand_silica_gel_plate_OK:=FALSE;
		展开工位允许放硅胶板:=FALSE;
		展开工位允许取硅胶板:=FALSE;
		展开工位机器人到达准备点:=FALSE;
		展开工位机器人放硅胶板完成:=FALSE;
		展开工位取硅胶板完成:=FALSE;
		展开工位允许放硅胶板1:=FALSE;
		CASE Expand_Group OF
			1:
				CASE Expand_Number OF
					1:
						展缸1气缸1手动:=FALSE;
						展缸1气缸1自动:=FALSE;
						展缸1进液电池阀1手动:=FALSE;
						展缸1进液电池阀1自动:=FALSE;
						展缸1排液电池阀1手动:=FALSE;
						展缸1排液电池阀1自动:=FALSE;
						展缸1吹气电池阀1手动:=FALSE;
						展缸1吹气电池阀1自动:=FALSE;
					2:
						展缸1气缸2手动:=FALSE;
						展缸1气缸2自动:=FALSE;
						展缸1进液电池阀2手动:=FALSE;
						展缸1进液电池阀2自动:=FALSE;
						展缸1排液电池阀2手动:=FALSE;
						展缸1排液电池阀2自动:=FALSE;
						展缸1吹气电池阀2手动:=FALSE;
						展缸1吹气电池阀2自动:=FALSE;	
					3:
						展缸1气缸3手动:=FALSE;
						展缸1气缸3自动:=FALSE;
						展缸1进液电池阀3手动:=FALSE;
						展缸1进液电池阀3自动:=FALSE;	
						展缸1排液电池阀3手动:=FALSE;
						展缸1排液电池阀3自动:=FALSE;
						展缸1吹气电池阀3手动:=FALSE;
						展缸1吹气电池阀3自动:=FALSE;	
					4:
						展缸1气缸4手动:=FALSE;
						展缸1气缸4自动:=FALSE;
						展缸1进液电池阀4手动:=FALSE;
						展缸1进液电池阀4自动:=FALSE;	
						展缸1排液电池阀4手动:=FALSE;
						展缸1排液电池阀4自动:=FALSE;
						展缸1吹气电池阀4手动:=FALSE;
						展缸1吹气电池阀4自动:=FALSE;	
				END_CASE
				IF %MW1300=0 AND 泵站位符=FALSE  THEN
					转发转存:='/1Z0,2,2R$R';     //泵初始化指令 
					%MW1300:=LEN(STR:= 转发转存);   //发送字节数
					泵站位符:=TRUE;
					初始化STEP:=10;
				END_IF
			2:
				CASE Expand_Number OF
					1:
						展缸2气缸1手动:=FALSE;
						展缸2气缸1自动:=FALSE;
						展缸2进液电池阀1手动:=FALSE;
						展缸2进液电池阀1自动:=FALSE;
						展缸2排液电池阀1手动:=FALSE;
						展缸2排液电池阀1自动:=FALSE;
						展缸2吹气电池阀1手动:=FALSE;
						展缸2吹气电池阀1自动:=FALSE;
					2:
						展缸2气缸2手动:=FALSE;
						展缸2气缸2自动:=FALSE;
						展缸2进液电池阀2手动:=FALSE;
						展缸2进液电池阀2自动:=FALSE;
						展缸2排液电池阀2手动:=FALSE;
						展缸2排液电池阀2自动:=FALSE;
						展缸2吹气电池阀2手动:=FALSE;
						展缸2吹气电池阀2自动:=FALSE;	
					3:
						展缸2气缸3手动:=FALSE;
						展缸2气缸3自动:=FALSE;
						展缸2进液电池阀3手动:=FALSE;
						展缸2进液电池阀3自动:=FALSE;	
						展缸2排液电池阀3手动:=FALSE;
						展缸2排液电池阀3自动:=FALSE;
						展缸2吹气电池阀3手动:=FALSE;
						展缸2吹气电池阀3自动:=FALSE;	
					4:
						展缸2气缸4手动:=FALSE;
						展缸2气缸4自动:=FALSE;
						展缸2进液电池阀4手动:=FALSE;
						展缸2进液电池阀4自动:=FALSE;	
						展缸2排液电池阀4手动:=FALSE;
						展缸2排液电池阀4自动:=FALSE;
						展缸2吹气电池阀4手动:=FALSE;
						展缸2吹气电池阀4自动:=FALSE;
				END_CASE 
				 IF %MW1300=0 AND 泵站位符=FALSE  THEN
					转发转存:='/2Z0,2,2R$R';     //泵初始化指令 
					%MW1300:=LEN(STR:= 转发转存);   //发送字节数
					泵站位符:=TRUE;
					初始化STEP:=10;
				END_IF
		END_CASE

		展开工位允许放硅胶板:=FALSE;
	
		
		
	10:
		CASE Expand_Group OF
			1:
				IF %MW1300=0 THEN
					转发转存:='/1Q$R';          //查询泵状态指令
					%MW1300:=LEN(STR:= 转发转存);
				END_IF
				
				
				IF R_TRIG[1].Q THEN
					泵初始化完成:=TRUE;
					泵站位符:=FALSE;
					初始化STEP:=0;
				END_IF
			2:
				IF %MW1300=0 THEN
					转发转存:='/2Q$R';          //查询泵状态指令
					%MW1300:=LEN(STR:= 转发转存);
				END_IF
				
				IF R_TRIG[2].Q THEN
					泵初始化完成:=TRUE;
					泵站位符:=FALSE;
					初始化STEP:=0;
				END_IF
		END_CASE
END_CASE
END_ACTION

ACTION A10_pipeline_cleaning_清洗管路:
TON[2](IN:=清洗STEP=10,PT:=T#1S);
TON_0(IN:=清洗STEP=20, PT:=T#3S , Q=> , ET=> );
R_TRIG[5](CLK:=%MX2005.5 , Q=> );  //泵空闲中
CASE 清洗STEP OF
	0 :
		大真空泵站位[10]:=TRUE;
		IF %MW1300=0 AND 泵站位符=FALSE  THEN
			转发转存:=Expand_forward_instructions; 
			%MW1300:=LEN(STR:= 转发转存);   //发送字节数
			泵站位符:=TRUE;
			清洗STEP:=10;
		END_IF
	10:
		//TON[2](IN:=TRUE,PT:=T#1S);
		IF %MW1300=0 AND TON[2].Q THEN
			CASE Expand_Group OF
				1:
					转发转存:='/1Q$R';          //查询泵状态指令
				2:
					转发转存:='/2Q$R';          //查询泵状态指令
			END_CASE
			%MW1300:=LEN(STR:= 转发转存);
		END_IF
		
		
		IF R_TRIG[5].Q THEN
			泵站位符:=FALSE;
			清洗STEP:=20;
		END_IF
	20:
		
		IF TON_0.Q THEN
			大真空泵站位[10]:=FALSE;
			转发转存:='';
			%MW1300:=128;
			Expand_Group_clean_OK:=TRUE;
			清洗STEP:=0;
		END_IF

		
END_CASE
END_ACTION

ACTION A20_clean_expand_润洗展缸:
TON[1](IN:=润洗展缸STEP=15,PT:=T#0.1S);
TON_1(IN:= 润洗展缸STEP=20  , PT:=T#5S , Q=> , ET=> );
TON_2(IN:=润洗展缸STEP=30, PT:=T#3S, Q=> , ET=> );
TON[4](IN:=润洗展缸STEP=40,PT:=T#30S);
TON[10](IN:=(Expand_Group=1 AND  展缸1溶剂废液检测传感器) OR (Expand_Group=2 AND  展缸2溶剂废液检测传感器),PT:=T#10S);
R_TRIG[3](CLK:=%MX2005.5 , Q=> );  //泵空闲中



CASE 润洗展缸STEP OF
	0 :
		润洗计数:=0;
		CASE Expand_Group OF
			1:
				CASE Expand_Number OF
					1:
						展缸1进液电池阀1自动:=TRUE;
						展缸1排液电池阀1自动:=TRUE;
						展缸1气缸1自动:=TRUE;
						润洗展缸STEP:=10;
					2:
						展缸1进液电池阀2自动:=TRUE;
						展缸1排液电池阀2自动:=TRUE;
						展缸1气缸2自动:=TRUE;
						润洗展缸STEP:=10;
					3:
						展缸1进液电池阀3自动:=TRUE;
						展缸1排液电池阀3自动:=TRUE;
						展缸1气缸3自动:=TRUE;
						润洗展缸STEP:=10;
					4:
						展缸1进液电池阀4自动:=TRUE;
						展缸1排液电池阀4自动:=TRUE;
						展缸1气缸4自动:=TRUE;
						润洗展缸STEP:=10;
				END_CASE
			
			2:
				CASE Expand_Number OF
					1:
						展缸2进液电池阀1自动:=TRUE;
						展缸2排液电池阀1自动:=TRUE;
						展缸2气缸1自动:=TRUE;
						润洗展缸STEP:=10;
					2:
						展缸2进液电池阀2自动:=TRUE;
						展缸2排液电池阀2自动:=TRUE;
						展缸2气缸2自动:=TRUE;
						润洗展缸STEP:=10;
					3:
						展缸2进液电池阀3自动:=TRUE;
						展缸2排液电池阀3自动:=TRUE;
						展缸2气缸3自动:=TRUE;
						润洗展缸STEP:=10;
					4:
						展缸2进液电池阀4自动:=TRUE;
						展缸2排液电池阀4自动:=TRUE;
						展缸2气缸4自动:=TRUE;
						润洗展缸STEP:=10;
				END_CASE
		END_CASE
	10:		
		IF %MW1300=0 AND 泵站位符=FALSE  THEN
			转发转存:=Expand_forward_instructions;   
			%MW1300:=LEN(STR:= 转发转存);   //发送字节数
			泵站位符:=TRUE;
			润洗展缸STEP:=15;
		END_IF
	15:
		
		IF %MW1300=0 AND TON[1].Q THEN
			CASE Expand_Group OF
				1:
					转发转存:='/1Q$R';           //查询泵状态指令
				2:
					转发转存:='/2Q$R';           //查询泵状态指令
			END_CASE
			%MW1300:=LEN(STR:= 转发转存);
		END_IF
		
		IF R_TRIG[3].Q THEN
			泵站位符:=FALSE;
			润洗计数:=润洗计数+1;
			IF 润洗计数>=Expand_rinse_count THEN
				润洗计数:=0;
				润洗展缸STEP:=20;
			ELSE
				润洗展缸STEP:=10;
			END_IF
			
		END_IF
		
	20:
		//TON_1(IN:= TRUE  , PT:=T#5S , Q=> , ET=> );
		IF TON_1.Q THEN
			转发转存:='';    
			%MW1300:=128;
			润洗展缸STEP:=30;
		END_IF
	30:
		//TON_2(IN:=TRUE, PT:=T#2S, Q=> , ET=> );
		IF TON_2.Q THEN
			大真空泵站位[9]:=TRUE;
			IF TON[10].Q THEN
				
				CASE Expand_Group OF
					1:
						CASE Expand_Number OF
							1:
								展缸1进液电池阀1自动:=FALSE;
								
								展缸1吹气电池阀1自动:=TRUE;
								
								
								润洗展缸STEP:=40;
							2:
								展缸1进液电池阀2自动:=FALSE;
								
								展缸1吹气电池阀2自动:=TRUE;
								
								
								润洗展缸STEP:=40;
							3:
								展缸1进液电池阀3自动:=FALSE;
								
								展缸1吹气电池阀3自动:=TRUE;
								
								
								润洗展缸STEP:=40;
							4:
								展缸1进液电池阀4自动:=FALSE;
								
								展缸1吹气电池阀4自动:=TRUE;
								
								润洗展缸STEP:=40;
						END_CASE
					
					2:
						CASE Expand_Number OF
							1:
								展缸2进液电池阀1自动:=FALSE;
								
								展缸2吹气电池阀1自动:=TRUE;
								
								润洗展缸STEP:=40;
							2:
								展缸2进液电池阀2自动:=FALSE;
								
								展缸2吹气电池阀2自动:=TRUE;
								
								润洗展缸STEP:=40;
							3:
								展缸2进液电池阀3自动:=FALSE;
								
								展缸2吹气电池阀3自动:=TRUE;
								
								润洗展缸STEP:=40;
							4:
								展缸2进液电池阀4自动:=FALSE;
								
								展缸2吹气电池阀4自动:=TRUE;
								润洗展缸STEP:=40;
						END_CASE
				END_CASE
			END_IF
		END_IF
	40:
		IF TON[4].Q THEN
			大真空泵站位[9]:=FALSE;
			CASE Expand_Group OF
				1:
					CASE Expand_Number OF
						1:
							展缸1排液电池阀1自动:=FALSE;
							展缸1吹气电池阀1自动:=FALSE;
							
							Expand_Group_clean_OK:=TRUE;
							润洗展缸STEP:=0;
						2:
							展缸1排液电池阀2自动:=FALSE;
							展缸1吹气电池阀2自动:=FALSE;
							
							Expand_Group_clean_OK:=TRUE;
							润洗展缸STEP:=0;
						3:
							展缸1排液电池阀3自动:=FALSE;
							展缸1吹气电池阀3自动:=FALSE;
							
							Expand_Group_clean_OK:=TRUE;
							润洗展缸STEP:=0;
						4:
							展缸1排液电池阀4自动:=FALSE;
							
							展缸1吹气电池阀4自动:=FALSE;
							Expand_Group_clean_OK:=TRUE;
							润洗展缸STEP:=0;
					END_CASE
				
				2:
					CASE Expand_Number OF
						1:
							展缸2排液电池阀1自动:=FALSE;
							展缸2吹气电池阀1自动:=FALSE;
							
							Expand_Group_clean_OK:=TRUE;
							润洗展缸STEP:=0;
						2:
							展缸2排液电池阀2自动:=FALSE;
							展缸2吹气电池阀2自动:=FALSE;
							
							Expand_Group_clean_OK:=TRUE;
							润洗展缸STEP:=0;
						3:
							展缸2排液电池阀2自动:=FALSE;
							展缸2吹气电池阀3自动:=FALSE;
							
							Expand_Group_clean_OK:=TRUE;
							润洗展缸STEP:=0;
						4:
							展缸2排液电池阀2自动:=FALSE;
							展缸2吹气电池阀4自动:=FALSE;
							
							Expand_Group_clean_OK:=TRUE;
							润洗展缸STEP:=0;
					END_CASE
			END_CASE
		END_IF
END_CASE
END_ACTION

ACTION A40_up_liquid_上液:
R_TRIG[6](CLK:=%MX2005.5 , Q=> );  //泵空闲中
TON[9](IN:=上液step=20,PT:=T#0.5S,);
IF Expand_Group>0 AND Expand_Number>0 THEN
	CASE 上液step OF
		0:
			CASE Expand_Group OF
				1:
					CASE Expand_Number OF
						1:
							展缸1进液电池阀1自动:=TRUE;
							上液step:=10;
						2:
							展缸1进液电池阀2自动:=TRUE;
							上液step:=10;
						3:
							展缸1进液电池阀3自动:=TRUE;
							上液step:=10;
						4:
							展缸1进液电池阀4自动:=TRUE;
							上液step:=10;
					END_CASE
				2:
					CASE Expand_Number OF
						1:
							展缸2进液电池阀1自动:=TRUE;
							上液step:=10;
						2:
							展缸2进液电池阀2自动:=TRUE;
							上液step:=10;
						3:
							展缸2进液电池阀3自动:=TRUE;
							上液step:=10;
						4:
							展缸2进液电池阀4自动:=TRUE;
							上液step:=10;
					END_CASE
			END_CASE
		10:
			IF %MW1300=0 AND 泵站位符=FALSE  THEN
				转发转存:=Expand_forward_instructions; 
				%MW1300:=LEN(STR:= 转发转存);   //发送字节数
				泵站位符:=TRUE;
				上液step:=20;
			END_IF
		20:
		
			IF %MW1300=0 AND TON[9].Q  THEN
				CASE Expand_Group OF
					 1:
						 转发转存:='/1Q$R';          //查询泵状态指令
					 2:
						 转发转存:='/2Q$R';          //查询泵状态指令
				END_CASE
				%MW1300:=LEN(STR:= 转发转存);
			END_IF
			
			
			IF R_TRIG[6].Q THEN
				泵站位符:=FALSE;
				转发转存:='';
				%MW1300:=128;
				上液计数:=上液计数+1;
				IF 上液计数>=Expand_up_liquid_count THEN
					上液计数:=0;
					CASE Expand_Group OF
						1:
							CASE Expand_Number OF
								1:
									展缸1进液电池阀1自动:=FALSE;
									;
								2:
									展缸1进液电池阀2自动:=FALSE;
									
								3:
									展缸1进液电池阀3自动:=FALSE;
									
								4:
									展缸1进液电池阀4自动:=FALSE;
									
							END_CASE
						2:
							CASE Expand_Number OF
								1:
									展缸2进液电池阀1自动:=FALSE;
									
								2:
									展缸2进液电池阀2自动:=FALSE;
									
								3:
									展缸2进液电池阀3自动:=FALSE;
									
								4:
									展缸2进液电池阀4自动:=FALSE;
									
							END_CASE
						END_CASE
					Expand_up_liquid_OK:=TRUE;
					上液step:=0;
				ELSE
					上液step:=10;
				END_IF
			END_IF	
    END_CASE	
END_IF
END_ACTION

ACTION A30_silica_gel_plate_放硅胶板:



CASE 放硅胶板step OF
	0:
		
		放硅胶板step:=10;
	10:
		展开工位允许放硅胶板1:=TRUE;
		IF 展开工位机器人到达准备点 THEN
			CASE Expand_Group OF
				1:
					CASE Expand_Number OF
						1:
							展缸1气缸1自动:=FALSE;
							IF 展缸1气缸1原点 THEN
								展开工位允许放硅胶板:=TRUE;
								ParameterList1:=1;
								放硅胶板step:=20;
							END_IF
							
						2:
							展缸1气缸2自动:=FALSE;
							IF 展缸1气缸2原点 THEN
								ParameterList1:=2;
								展开工位允许放硅胶板:=TRUE;
								放硅胶板step:=20;
							END_IF
						3:
							展缸1气缸3自动:=FALSE;
							IF 展缸1气缸3原点 THEN
								ParameterList1:=3;
								展开工位允许放硅胶板:=TRUE;
								放硅胶板step:=20;
							END_IF
						4:
							展缸1气缸4自动:=FALSE;
							IF 展缸1气缸4原点 THEN
								ParameterList1:=4;
								展开工位允许放硅胶板:=TRUE;
								放硅胶板step:=20;
							END_IF
					END_CASE
				2:
					CASE Expand_Number OF
						1:
							展缸2气缸1自动:=FALSE;
							IF 展缸2气缸1原点 THEN
								ParameterList1:=5;
								展开工位允许放硅胶板:=TRUE;
								放硅胶板step:=20;
							END_IF
						2:
							展缸2气缸2自动:=FALSE;
							IF 展缸2气缸2原点 THEN
								ParameterList1:=6;
								展开工位允许放硅胶板:=TRUE;
								放硅胶板step:=20;
							END_IF
						3:
							展缸2气缸3自动:=FALSE;
							IF 展缸2气缸3原点 THEN
								ParameterList1:=7;
								展开工位允许放硅胶板:=TRUE;
								放硅胶板step:=20;
							END_IF
						4:
							展缸2气缸4自动:=FALSE;
							IF 展缸2气缸4原点 THEN
								ParameterList1:=8;
								展开工位允许放硅胶板:=TRUE;
								放硅胶板step:=20;
							END_IF
					END_CASE
			END_CASE	
		END_IF
	20:
		IF 展开工位机器人放硅胶板完成 THEN
			展开工位允许放硅胶板:=FALSE;
			展开工位允许放硅胶板1:=FALSE;
			CASE Expand_Group OF
				1:
					CASE Expand_Number OF
						1:
							展缸1气缸1自动:=TRUE ;
							IF 展缸1气缸1动点 THEN
								放硅胶板step:=30;
							END_IF
							
						2:
							展缸1气缸2自动:=TRUE;
							IF 展缸1气缸2动点 THEN
								
								放硅胶板step:=30;
							END_IF
						3:
							展缸1气缸3自动:=TRUE;
							IF 展缸1气缸3动点 THEN
								
								放硅胶板step:=30;
							END_IF
						4:
							展缸1气缸4自动:=TRUE ;
							IF 展缸1气缸4动点 THEN
								
								放硅胶板step:=30;
							END_IF
					END_CASE
				2:
					CASE Expand_Number OF
						1:
							展缸2气缸1自动:=TRUE;
							IF 展缸2气缸1动点 THEN
								
								放硅胶板step:=30;
							END_IF
						2:
							展缸2气缸2自动:=TRUE ;
							IF 展缸2气缸2动点 THEN
								
								放硅胶板step:=30;
							END_IF
						3:
							展缸2气缸3自动:=TRUE;
							IF 展缸2气缸3动点 THEN
								
								放硅胶板step:=30;
							END_IF
						4:
							展缸2气缸4自动:=TRUE;
							IF 展缸2气缸4动点 THEN
								
								放硅胶板step:=30;
							END_IF
					END_CASE
			END_CASE	
		END_IF
	30:
		展开工位机器人放硅胶板完成:=FALSE;
		Expand_silica_gel_plate_OK:=TRUE;
		放硅胶板step:=0;
	
	
	

END_CASE
END_ACTION

END_PROGRAM

// Device/Application/40_Man/Robotic_Process_机器人流程
PROGRAM Robotic_Process_机器人流程
VAR
	RB_Control_0: FB_RB_Control;
	
	TON: TON;
	R_TRIG: ARRAY[1..2] OF R_TRIG;
END_VAR


R_TRIG[1](CLK:=collect_Old_Plate_Slot>0);
R_TRIG[2](CLK:=scrape_Old_Plate_Slot>0);
//机器人流程
IF MODE_State=1 THEN	
	IF R_TRIG[1].Q THEN
		收集瓶组站位符:=TRUE;
	END_IF
	IF R_TRIG[2].Q THEN
		收集器组站位符:=TRUE;
	END_IF

	CASE 机器人流程 OF
		0:
			IF Status=0 THEN
				IF 上样点样允许放硅胶板 THEN
					机器人流程:=10;
				ELSIF  上样点样允许取硅胶板 AND scrape_Step=0 AND NOT 刮板拍照工位站位符 THEN 
					机器人流程:=20;
				ELSIF 拍照工位允许取硅胶板去展开 AND (Expand_Step=0 OR Expand_Step=30) THEN
					机器人流程:=30;
				ELSIF 展开工位允许取硅胶板 AND scrape_Step=0 AND NOT 刮板拍照工位站位符 THEN       //刮板拍照空闲
					机器人流程:=40;
				ELSIF scrape_Fetch_Rack_Plate>0 AND NOT 刮板拍照暂存工位传感器 THEN 
					机器人流程:=70;
				ELSIF collect_Fetch_Rack_Plate>0 AND NOT 收集平台暂存工位传感器 THEN
					机器人流程:=60;
				ELSIF collect_Old_Plate_Slot>0 AND 收集平台暂存工位传感器 AND NOT 收集瓶组站位符  THEN
					机器人流程:=80;
				ELSIF scrape_Old_Plate_Slot>0 AND 刮板拍照暂存工位传感器 AND  NOT 收集器组站位符 THEN
					机器人流程:=90;
				ELSIF 拍照工位允许放收集器 AND 刮板拍照暂存工位传感器 AND scrape_Consume_Slot>0 THEN 
					机器人流程:=100;
				ELSIF 拍照工位允许取收集器 AND collect_Step=0 THEN           //收集工位空闲
					机器人流程:=110;
				ELSIF 收集工位允许放收集瓶 AND 收集平台暂存工位传感器 AND collect_Consume_Slot>0 THEN
					机器人流程:=120;
				ELSIF 收集工位允许取收集器 AND collect_Powder_Return_Slot>0 THEN
					机器人流程:=130;
				ELSIF 收集工位允许机器人取收集瓶放暂存工位 AND collect_Consume_Slot>0 THEN
					机器人流程:=140;
				ELSIF 拍照工位允许取硅胶板放废料区 THEN
					机器人流程:=50;
				END_IF
			END_IF
			

	
//	取升降机硅胶板放点样机构上

		10:                                                  
			ParameterList3:=1;                           //取1号吸盘工具
			A00_取放工具();
			IF 取工具完成 THEN
				取工具完成:=FALSE;
				ParameterList3:=0; 
				机器人流程:=11;
			END_IF
		11:
			A10_取升降机硅胶板();
			IF 取升降硅胶板完成 THEN
				取升降硅胶板完成:=FALSE;
				机器人流程:=12;		
			END_IF
		12:
			A15_放点样硅胶板();
			IF 放点样硅胶板完成 THEN
				FunctionID:=0;
				放点样硅胶板完成:=FALSE;
				机器人流程:=0;
			END_IF
			
				




//取点样硅胶板放拍照机构上
		20:
			ParameterList3:=1;                           //取1号吸盘工具
			A00_取放工具();
			IF 取工具完成 THEN
				取工具完成:=FALSE;
				机器人流程:=21;
			END_IF
		21:
			A20_取点样硅胶板();
			IF 取点样硅胶板完成 THEN
				
				机器人流程:=22;
			END_IF
		22:
			IF 拍照工位允许放硅胶板 THEN
				
				机器人流程:=23;
			END_IF
		23:
			A35_放拍照硅胶板();
			IF 放拍照硅胶板完成 THEN
				FunctionID:=0;
				放拍照硅胶板完成:=FALSE;
				机器人流程:=0;
			END_IF




//取拍照机构硅胶板放展缸
		30:
			ParameterList3:=1;                           //取1号吸盘工具
			A00_取放工具();
			IF 取工具完成 THEN
				取工具完成:=FALSE;
				机器人流程:=31;
			END_IF
		31:
			A32_取拍照硅胶板();
			IF 取拍照硅胶板完成 THEN
				
				机器人流程:=32;
			END_IF
		32:
			IF 展开工位允许放硅胶板1 THEN
				机器人流程:=33;
			END_IF
		33:
			A25_放展缸硅胶板();
			IF 展开工位机器人放硅胶板完成 THEN
				FunctionID:=0;
				机器人流程:=0;
			END_IF
				
				



//取展缸硅胶板到拍照刮取机构
		40:
			ParameterList3:=1;                           //取1号吸盘工具
			A00_取放工具();
			IF 取工具完成 THEN
				取工具完成:=FALSE;
				机器人流程:=41;
			END_IF
		41:
			A30_取展缸硅胶板();
			IF 取展缸硅胶板完成 THEN
				取展缸硅胶板完成:=FALSE;
				展开工位允许取硅胶板:=FALSE;
				机器人流程:=42;
			END_IF
		42:
			IF 拍照工位允许放硅胶板 THEN
				机器人流程:=43;
			END_IF
		43:
			A35_放拍照硅胶板();
			IF 放拍照硅胶板完成 THEN
				FunctionID:=0;
				放拍照硅胶板完成:=FALSE;
				机器人流程:=0;
			END_IF
			
			





//取拍照刮取硅胶板放到废料区
		50:
			ParameterList3:=1;                           //取1号吸盘工具
			A00_取放工具();
			IF 取工具完成 THEN
				取工具完成:=FALSE;
				机器人流程:=51;
			END_IF
		51:
			A32_取拍照硅胶板();
			IF 取拍照硅胶板完成 THEN
				取拍照硅胶板完成:=FALSE;
				机器人流程:=52;
			END_IF
		52:
			A65_放废料硅胶板();
			IF 取刮板硅胶板放废料区完成 THEN
				拍照工位允许取硅胶板放废料区:=FALSE;
				取刮板硅胶板放废料区完成:=FALSE;
				FunctionID:=0;
				
				机器人流程:=0;
			END_IF







//取收集瓶组到暂存工位
		60:
			ParameterList3:=2;            //取2号大夹持工具
			A00_取放工具();
			IF 取工具完成 THEN
				取工具完成:=FALSE;
				机器人流程:=61;
			END_IF
		61:
			A41_取收集瓶组放暂存工位();
			IF 取收集瓶组放暂存工位完成 THEN
				collect_Fetch_Rack_Plate:=0;
				FunctionID:=0;
				机器人流程:=0;
				取收集瓶组放暂存工位完成:=FALSE;
			END_IF
			
			





//取收集器组到暂存工位
		70:
			ParameterList3:=2;            //取2号大夹持工具
			A00_取放工具();
			IF 取工具完成 THEN
				取工具完成:=FALSE;
				机器人流程:=71;
			END_IF
		71:
			A40_取收集器组放暂存工位();
			IF 取收集器组放暂存工位完成 THEN
				scrape_Fetch_Rack_Plate:=0;
				FunctionID:=0;
				机器人流程:=0;
				取收集器组放暂存工位完成:=FALSE;
			END_IF
		
		
		
		
		
//取收集瓶暂存工位到仓库
		80:
			ParameterList3:=2;            //取2号大夹持工具
			A00_取放工具();
			IF 取工具完成 THEN
				取工具完成:=FALSE;
				机器人流程:=81;
			END_IF
		81:
			A71_取暂存收集瓶放仓库();
			IF 取暂存收集瓶组放仓库完成 THEN
				collect_Old_Plate_Slot:=0;
				FunctionID:=0;
				机器人流程:=0;
				取暂存收集瓶组放仓库完成:=FALSE;
			END_IF		
		
		
		
		
		
	
	
	


//取收集器暂存工位到仓库
		90:
			ParameterList3:=2;            //取2号大夹持工具
			A00_取放工具();
			IF 取工具完成 THEN
				取工具完成:=FALSE;
				机器人流程:=91;
			END_IF
		91:
			A70_取暂存收集器组放仓库();
			IF 取暂存收集器组放仓库完成 THEN
				scrape_Old_Plate_Slot:=0;
				FunctionID:=0;
				机器人流程:=0;
				取暂存收集器组放仓库完成:=FALSE;
			END_IF	







//取暂存收集器到刮取位
		100:
			ParameterList3:=3;                           //取3号小夹持工具
			A00_取放工具();
			IF 取工具完成 THEN
				取工具完成:=FALSE;
				机器人流程:=101;
			END_IF	
		101:
			A45_取暂存收集器放刮板位();
			IF 取暂存收集器放刮板位完成 THEN
				scrape_Consume_Slot:=0;
				FunctionID:=0;
				取暂存收集器放刮板位完成:=FALSE;
				机器人流程:=0;
			END_IF
			
			






//取刮板拍照收集器到收集工位
		110:
			ParameterList3:=3;                           //取3号小夹持工具
			A00_取放工具();
			IF 取工具完成 THEN
				取工具完成:=FALSE;
				机器人流程:=111;
			END_IF
		111:
			A55_取刮板收集器放到收集工位();
			IF 取刮板收集器放到收集工位完成 THEN
				FunctionID:=0;
				取刮板收集器放到收集工位完成:=FALSE;
				机器人流程:=0;
			END_IF
			
	
	
	
	
	
	
	
//取暂存收集瓶到收集工位	
		120:
			ParameterList3:=3;                           //取3号小夹持工具
			A00_取放工具();
			IF 取工具完成 THEN
				取工具完成:=FALSE;
				机器人流程:=121;
			END_IF
		121:
			A50_取暂存收集瓶放收集工位();
			IF 取暂存收集瓶放收集工位完成 THEN
				FunctionID:=0;
				取暂存收集瓶放收集工位完成:=FALSE;
				机器人流程:=0;
			END_IF
			
			






//取收集器到暂存工位
		130:
			ParameterList3:=3;                           //取3号小夹持工具
			A00_取放工具();
			IF 取工具完成 THEN
				取工具完成:=FALSE;
				机器人流程:=131;
			END_IF
		131:
			A60_取收集器放暂存工位();
			IF 取收集器放暂存工位完成 THEN
				collect_Powder_Return_Slot:=0;
				收集器组站位符:=FALSE;
				收集工位放收集器完成:=TRUE;
				FunctionID:=0;
				机器人流程:=0;
				取收集器放暂存工位完成:=FALSE;
			END_IF
			
			




//取收集瓶到暂存工位
		140:
			ParameterList3:=3;                           //取3号小夹持工具
			A00_取放工具();
			IF 取工具完成 THEN
				取工具完成:=FALSE;
				机器人流程:=141;
			END_IF
		141:
			A65_取收集瓶放暂存工位();
			IF 取收集瓶放暂存工位完成 THEN
				scrape_Consume_Slot:=0;
				收集瓶组站位符:=FALSE;
				FunctionID:=0;
				机器人流程:=0;
				取收集瓶放暂存工位完成:=FALSE;
			END_IF
			


    END_CASE
END_IF

ACTION A30_取展缸硅胶板:




CASE 取展缸硅胶板step OF
	0:
		地轨轴11YDATE.fAbsTarget:=HMI_地轨轴11Y.position[5];     //地轨去展开位
		地轨轴11YDATE.xMoveAbs:=TRUE;
		IF 地轨轴11YDATE.bAbMoveDone THEN
			地轨轴11YDATE.xMoveAbs:=FALSE;
			取展缸硅胶板step:=10;
		END_IF
	10:
		IF  ParameterList1>0 AND Status=0 THEN
			FunctionID:=5;                                  //取展缸硅胶板
			Execute:=1;
			取展缸硅胶板step:=20;
		END_IF
	20:
		IF RO_ParameterList1>0 AND Status=2 THEN                       //取硅胶板完成
			Execute:=0;
			取展缸硅胶板完成:=TRUE;
			取展缸硅胶板step:=0;
		END_IF
END_CASE
END_ACTION

ACTION A60_取收集器放暂存工位:


CASE 取收集器放暂存工位step OF
	0:
		地轨轴11YDATE.fAbsTarget:=HMI_地轨轴11Y.position[3];     //地轨去取收集组位置暂存位置
			地轨轴11YDATE.xMoveAbs:=TRUE;
			取收集器放暂存工位step:=5;
			
	5:
		IF 地轨轴11YDATE.bAbMoveDone  THEN
			地轨轴11YDATE.xMoveAbs:=FALSE;
			FunctionID:=12;  
			ParameterList8:=6;                               //放收集器回暂存工位
			Execute:=1;
			取收集器放暂存工位step:=10;
		END_IF
	10:
		IF RO_ParameterList8=6  THEN                       //放收集器回暂存工位完成
			收集工位机器人到达收集器位置:=TRUE;
			取收集器放暂存工位step:=30;
		END_IF
	30:
		IF 收集工位机器人取收集器放回暂存工位 THEN
			ParameterList8:=7;                               //机器人去取收集器
			ParameterList7:=collect_Powder_Return_Slot;
			收集工位机器人取收集器放回暂存工位:=FALSE;
			取收集器放暂存工位step:=40;
		END_IF
	40:
		IF RO_ParameterList8=7 AND Status=2 THEN                         //到达夹持位置
			Execute:=0;
			取收集器放暂存工位完成:=TRUE;
			取收集器放暂存工位step:=0;
		END_IF
END_CASE
END_ACTION

ACTION A00_取放工具:



CASE 取工具setp OF
	0:
		IF RO_ParameterList3=ParameterList3 THEN
			取工具完成:=TRUE;
			取工具setp:=0;
		ELSE
			取工具setp:=5;
		END_IF
	5:
		地轨轴11YDATE.fAbsTarget:=HMI_地轨轴11Y.position[4];     //地轨去取工具位置
		地轨轴11YDATE.xMoveAbs:=TRUE;
		IF 地轨轴11YDATE.bAbMoveDone THEN
			地轨轴11YDATE.xMoveAbs:=FALSE;
			FunctionID:=23;                              //取工具ID
			Execute:=1;                                  //机器人启动                        
			取工具setp:=10;
		END_IF
	10:
		IF RO_ParameterList3=ParameterList3 AND Status=2 THEN                               //取工具完成                                   
			Execute:=0;
			取工具完成:=TRUE;
			取工具setp:=0;
		END_IF
END_CASE
END_ACTION

ACTION A35_放拍照硅胶板:




CASE 放拍照硅胶板step OF
	0:
		地轨轴11YDATE.fAbsTarget:=HMI_地轨轴11Y.position[2];     //地轨去刮板拍照位
		地轨轴11YDATE.xMoveAbs:=TRUE;
		IF 地轨轴11YDATE.bAbMoveDone AND Status=0 THEN
				地轨轴11YDATE.xMoveAbs:=FALSE;
				FunctionID:=6;                              //放拍照硅胶板
				ParameterList5:=1;                           //放硅胶板到刮板拍照位
				Execute:=1;                                  //机器人启动                        
				放拍照硅胶板step:=10;
		END_IF
	10:
		IF RO_ParameterList5=1 AND Status=2 THEN              //放硅胶板完成
			Execute:=0; 
			ParameterList5:=0;
			拍照工位放硅胶板完成:=TRUE;
			放拍照硅胶板完成:=TRUE;
			放拍照硅胶板step:=0;
		END_IF
END_CASE
END_ACTION

ACTION A65_放废料硅胶板:



CASE 取刮板硅胶板放废料区step OF
	0:
		地轨轴11YDATE.fAbsTarget:=HMI_地轨轴11Y.position[1];     //地轨去上样点样位置
			地轨轴11YDATE.xMoveAbs:=TRUE;
			IF 地轨轴11YDATE.bAbMoveDone THEN
				地轨轴11YDATE.xMoveAbs:=FALSE;
				取刮板硅胶板放废料区step:=5;
            END_IF
	5:
		IF  升降下料伺服允许放料 AND  Status=0 THEN
			
			FunctionID:=8; 
			ParameterList4:=3;                                     //机器人放到废料区
			Execute:=1; 
			取刮板硅胶板放废料区step:=10;
		END_IF
	10:
		IF RO_ParameterList4=3 AND Status=2  THEN                               //机器人放废料区完成
			Execute:=0; 
			刮板拍照工位站位符:=FALSE;
			升降下料机器人放废料完成:=TRUE;
			取刮板硅胶板放废料区完成:=TRUE;
			取刮板硅胶板放废料区step:=0;
		END_IF
END_CASE
END_ACTION

ACTION A41_取收集瓶组放暂存工位:


CASE 取收集瓶组放暂存工位step OF
	0:
			地轨轴11YDATE.fAbsTarget:=HMI_地轨轴11Y.position[6];     //地轨去取收集组位置
			地轨轴11YDATE.xMoveAbs:=TRUE;
			溶液收集瓶定位自动:=FALSE;
			取收集瓶组放暂存工位step:=10;
	10:
		IF 地轨轴11YDATE.bAbMoveDone AND Status=0 THEN
				地轨轴11YDATE.xMoveAbs:=FALSE;
				FunctionID:=21;                              //取收集瓶组
				ParameterList6:=collect_Fetch_Rack_Plate+6;       //取收集瓶组坐标
				Execute:=1;                                  //机器人启动                        
				取收集瓶组放暂存工位step:=20;
			END_IF
	20:
		IF RO_ParameterList6=ParameterList6 AND Status=2 THEN             //取收集瓶组完成
			Execute:=0;
			地轨轴11YDATE.fAbsTarget:=HMI_地轨轴11Y.position[3];     //地轨去收集工位
			地轨轴11YDATE.xMoveAbs:=TRUE;
			取收集瓶组放暂存工位step:=30;
		END_IF
	30:
		IF 地轨轴11YDATE.bAbMoveDone AND Status=0 THEN
				地轨轴11YDATE.xMoveAbs:=FALSE;
				FunctionID:=22;                              //放收集瓶组
				ParameterList6:=14;                         //放收集瓶组
				Execute:=1;                                  //机器人启动                        
				取收集瓶组放暂存工位step:=40;
		END_IF
	40:
		IF RO_ParameterList6=14 AND Status=2 THEN                        //放收集瓶完成
			Execute:=0; 
			ParameterList6:=0;
			溶液收集瓶定位自动:=TRUE;
			取收集瓶组放暂存工位完成:=TRUE;
			取收集瓶组放暂存工位step:=0;
		END_IF
END_CASE
END_ACTION

ACTION A40_取收集器组放暂存工位:




CASE 取收集器组放暂存工位step OF
	0:
		地轨轴11YDATE.fAbsTarget:=HMI_地轨轴11Y.position[6];     //地轨去取收集组位置
		地轨轴11YDATE.xMoveAbs:=TRUE;
		取收集器组放暂存工位step:=10;
	
	10:
		IF 地轨轴11YDATE.bAbMoveDone  AND Status=0 THEN
				地轨轴11YDATE.xMoveAbs:=FALSE;
				FunctionID:=19;                              //取收集器组
				ParameterList6:=scrape_Fetch_Rack_Plate;       //取收集器组坐标
				Execute:=1;                                  //机器人启动                        
				取收集器组放暂存工位step:=20;
			END_IF
	20:
		IF RO_ParameterList6=ParameterList6 AND Status=2 THEN             //取收集器组完成
			Execute:=0;
			地轨轴11YDATE.fAbsTarget:=HMI_地轨轴11Y.position[3];     //地轨去收集
			地轨轴11YDATE.xMoveAbs:=TRUE;
			取收集器组放暂存工位step:=30;
		END_IF
	30:
		IF 地轨轴11YDATE.bAbMoveDone AND Status=0 THEN
				地轨轴11YDATE.xMoveAbs:=FALSE;
				FunctionID:=20;                              //放收集器组
				ParameterList6:=13;                         //取收集器组坐标
				Execute:=1;                                  //机器人启动                        
				取收集器组放暂存工位step:=40;
		END_IF
	40:
		IF RO_ParameterList6=13  AND Status=2 THEN                        //放收集器完成
			Execute:=0; 
			粉末收集器定位自动:=TRUE;
			取收集器组放暂存工位完成:=TRUE;
			取收集器组放暂存工位step:=0;
		END_IF
	
END_CASE
END_ACTION

ACTION A15_放点样硅胶板:



CASE 放点样硅胶板step OF
	0:	IF  Status=0 THEN
	  		ParameterList4:=0;
			FunctionID:=2;                         //放点样硅胶板
			ParameterList2:=1;                     //机器人放硅胶板
			Execute:=1;
			放点样硅胶板step:=10;
	  	END_IF
		
	10:
		IF RO_ParameterList2=1 AND Status=2 THEN         //机器人放硅胶板完成
			上样点样放硅胶板完成:=TRUE;
			Execute:=0;
			放点样硅胶板完成:=TRUE;
			放点样硅胶板step:=0;
		END_IF
END_CASE
END_ACTION

ACTION A55_取刮板收集器放到收集工位:



CASE 取刮板收集器放到收集工位step OF
	0:
		地轨轴11YDATE.fAbsTarget:=HMI_地轨轴11Y.position[2];     //地轨去取收集组位置暂存位置
			地轨轴11YDATE.xMoveAbs:=TRUE;
			取刮板收集器放到收集工位step:=1;
	1:
		IF 地轨轴11YDATE.bAbMoveDone AND 拍照工位允许取收集器 AND  Status=0 THEN
			地轨轴11YDATE.xMoveAbs:=FALSE;
			拍照工位机器人退出工位完成:=FALSE;
			FunctionID:=11;
			Execute:=1;
			ParameterList5:=4;                          //机器人去夹持工位
			取刮板收集器放到收集工位step:=10;
		END_IF
	10:
		IF RO_ParameterList5=4 THEN
			拍照工位机器人到达收集器夹持位:=TRUE;
			取刮板收集器放到收集工位step:=20;
		END_IF
	20:
		IF 拍照工位机器人退出 THEN
			
			拍照工位机器人到达收集器夹持位:=FALSE;
			ParameterList5:=5;                          //机器人退出工位
			取刮板收集器放到收集工位step:=30;
		END_IF
	30:
		IF RO_ParameterList5=5 THEN
			拍照工位机器人退出完成:=TRUE;
			Execute:=0;
			地轨轴11YDATE.fAbsTarget:=HMI_地轨轴11Y.position[3];     //地轨去收集工位
			地轨轴11YDATE.xMoveAbs:=TRUE;
			取刮板收集器放到收集工位step:=40;
		END_IF
	40:
		IF 地轨轴11YDATE.bAbMoveDone THEN
			地轨轴11YDATE.xMoveAbs:=FALSE;                     
			取刮板收集器放到收集工位step:=50;
		END_IF
	50:
		IF 收集工位允许放收集器 AND  Status=0 THEN
			FunctionID:=12;                             //放收集工位收集器
			ParameterList8:=1;                         //机器人放收集器到夹持工位
			Execute:=1;
			取刮板收集器放到收集工位step:=60;
		END_IF
	60:
		IF RO_ParameterList8=1 THEN
			
			收集工位放收集器到工位:=TRUE;
			取刮板收集器放到收集工位step:=70;
		END_IF
	70:
		IF 收集工位允许机器人退出工位 THEN
			ParameterList8:=2;                     //机器人退出工位
			取刮板收集器放到收集工位step:=80;
		END_IF
	80:
		IF RO_ParameterList8=2 AND Status=2 THEN                //机器人退出工位完成
			Execute:=0;
			收集工位机器人退出完成:=TRUE;
			收集工位放收集器到工位:=FALSE;
			取刮板收集器放到收集工位完成:=TRUE;
			取刮板收集器放到收集工位step:=0;
		END_IF
END_CASE
END_ACTION

ACTION A45_取暂存收集器放刮板位:


CASE 取暂存收集器放刮板位step OF
	0:
		IF RO_ParameterList3=3 THEN
			ParameterList3:=0;
			Execute:=0;
			地轨轴11YDATE.fAbsTarget:=HMI_地轨轴11Y.position[2];     //地轨去刮板拍照位
			地轨轴11YDATE.xMoveAbs:=TRUE;
			取暂存收集器放刮板位step:=10;
		END_IF
	10:
		IF 地轨轴11YDATE.bAbMoveDone THEN
			地轨轴11YDATE.xMoveAbs:=FALSE;                     
			取暂存收集器放刮板位step:=20;
		END_IF
	20:
		IF 拍照工位允许放收集器 AND Status=0 THEN
			FunctionID:=9;                              //取暂存收集器
			ParameterList7:=scrape_Consume_Slot;           //取收集器
			Execute:=1;
			取暂存收集器放刮板位step:=30;
		END_IF
	30:
		IF RO_ParameterList7=ParameterList7  THEN                   //取收集器完成
			Execute:=0;
			取暂存收集器放刮板位step:=40;
		END_IF
	40:
		IF Status=0 THEN
			FunctionID:=10;                             //放收集器
			ParameterList5:=2;                         //机器人放收集器到夹持工位
			Execute:=1;
			取暂存收集器放刮板位step:=45;
		END_IF
	45:
		IF RO_ParameterList5=2 THEN
			拍照工位机器人到达夹持位:=TRUE;
			取暂存收集器放刮板位step:=50;
		END_IF
	50:
		IF 拍照工位机器人退出工位 THEN
			ParameterList5:=3;                         //机器人退出工位
			拍照工位机器人到达夹持位:=FALSE;
			取暂存收集器放刮板位step:=60;
		END_IF
	60:
		IF RO_ParameterList5=3 AND Status=2 THEN                    //机器人退出工位完成
			Execute:=0;
			拍照工位机器人退出工位完成:=TRUE;
			取暂存收集器放刮板位完成:=TRUE;
			取暂存收集器放刮板位step:=0;
		END_IF	
	
	
	
	
END_CASE
END_ACTION

ACTION A20_取点样硅胶板:



CASE 取点样硅胶板step OF
	0:
		地轨轴11YDATE.fAbsTarget:=HMI_地轨轴11Y.position[1];     //地轨去上样点样位置
			地轨轴11YDATE.xMoveAbs:=TRUE;
			IF 地轨轴11YDATE.bAbMoveDone THEN
				地轨轴11YDATE.xMoveAbs:=FALSE; 
				取点样硅胶板step:=5;
			END_IF
	5:
		IF  Status=0 THEN    //上样点样完成，展开准备完成
			FunctionID:=3;                              //取点样硅胶板
			ParameterList2:=2;                          //取硅胶板参数
			Execute:=1;                                  //机器人启动                        
			取点样硅胶板step:=10;
		END_IF
	10:
		IF RO_ParameterList2=2 AND Status=2 THEN
			Execute:=0;
			ParameterList2:=0;
			上样点样允许取硅胶板:=FALSE;
			取点样硅胶板完成:=TRUE;
			取点样硅胶板step:=0;
		END_IF
END_CASE
END_ACTION

ACTION A25_放展缸硅胶板:



CASE 放展缸硅胶板step OF
	0:	
		地轨轴11YDATE.fAbsTarget:=HMI_地轨轴11Y.position[5];     //地轨去展开位
		地轨轴11YDATE.xMoveAbs:=TRUE;
		IF 地轨轴11YDATE.bAbMoveDone AND Status=0 THEN
			地轨轴11YDATE.xMoveAbs:=FALSE;
			展开工位机器人到达准备点:=TRUE;
			放展缸硅胶板step:=5;
		END_IF
	5:
		IF 展开工位允许放硅胶板 THEN
			FunctionID:=4;                              //放展缸硅胶板
			Execute:=1;                                  //机器人启动       
			展开工位机器人到达准备点:=FALSE;
			放展缸硅胶板step:=10;
		END_IF
			
	10:
		IF RO_ParameterList1>0 AND Status=2 THEN                       //放硅胶板完成
			展开工位机器人放硅胶板完成:=TRUE;
			FunctionID:=0;
			Execute:=0;
			放展缸硅胶板step:=0;
		END_IF
END_CASE
END_ACTION

ACTION A50_取暂存收集瓶放收集工位:




CASE 取暂存收集瓶放收集工位step OF
	0:
		地轨轴11YDATE.fAbsTarget:=HMI_地轨轴11Y.position[3];     //地轨去取收集组位置暂存位置
			地轨轴11YDATE.xMoveAbs:=TRUE;
			取暂存收集瓶放收集工位step:=1;
	1:
		IF 地轨轴11YDATE.bAbMoveDone AND Status=0 THEN
			地轨轴11YDATE.xMoveAbs:=FALSE;
			FunctionID:=13;                             //取收集瓶
			ParameterList9:=collect_Consume_Slot;           //取收集瓶参数
			Execute:=1;
			取暂存收集瓶放收集工位step:=5;
		END_IF
	5:
		IF RO_ParameterList9=ParameterList9 AND 收集工位允许放收集瓶 THEN        //取收集瓶完成
			Execute:=0;
			取暂存收集瓶放收集工位step:=6;
		END_IF
	6:
		IF Status=0 THEN
			FunctionID:=15;  
			ParameterList8:=3;
			Execute:=1;
			取暂存收集瓶放收集工位step:=10;
		END_IF
	10:
		IF RO_ParameterList8=3 AND Status=2 THEN
				Execute:=0;
			收集工位放收集瓶完成:=TRUE;
			取暂存收集瓶放收集工位完成:=TRUE;
			取暂存收集瓶放收集工位step:=0;
		END_IF
END_CASE
END_ACTION

ACTION A71_取暂存收集瓶放仓库:






CASE 取暂存收集瓶组放仓库step OF
	0:
		地轨轴11YDATE.fAbsTarget:=HMI_地轨轴11Y.position[3];     //地轨去取收集组位置暂存位置
		地轨轴11YDATE.xMoveAbs:=TRUE;
		溶液收集瓶定位自动:=FALSE;
		取暂存收集瓶组放仓库step:=10;
	10:
		IF 地轨轴11YDATE.bAbMoveDone AND  Status=0 THEN
			地轨轴11YDATE.xMoveAbs:=FALSE;
			FunctionID:=14;                              //放收集器/瓶到仓库
			ParameterList6:=16;                          //取暂存收集器组
			Execute:=1; 
			取暂存收集瓶组放仓库step:=20;
		END_IF
	20:
		IF RO_ParameterList6=16 AND Status=2 THEN                      //取完成
			Execute:=0; 
			地轨轴11YDATE.fAbsTarget:=HMI_地轨轴11Y.position[6];     //地轨去放收集组位置
			地轨轴11YDATE.xMoveAbs:=TRUE;
			取暂存收集瓶组放仓库step:=30;
		END_IF
	30:
		IF 地轨轴11YDATE.bAbMoveDone AND Status=0 THEN
			地轨轴11YDATE.xMoveAbs:=FALSE;
			ParameterList6:=collect_Old_Plate_Slot+6;               //取暂存收集瓶组
			Execute:=1; 
			取暂存收集瓶组放仓库step:=40;
		END_IF
	40:
		IF RO_ParameterList6=collect_Old_Plate_Slot+6  AND Status=2 THEN
			取暂存收集瓶组放仓库完成:=TRUE;
			Execute:=0; 
			取暂存收集瓶组放仓库step:=0;
		END_IF
END_CASE
END_ACTION

ACTION A65_取收集瓶放暂存工位:

CASE 取收集瓶放暂存工位step OF
	0:
		地轨轴11YDATE.fAbsTarget:=HMI_地轨轴11Y.position[3];     //地轨去取收集组位置暂存位置
			地轨轴11YDATE.xMoveAbs:=TRUE;
			取收集瓶放暂存工位step:=5;
	5:
		IF 地轨轴11YDATE.bAbMoveDone AND 收集工位允许机器人取收集瓶放暂存工位 THEN
			地轨轴11YDATE.xMoveAbs:=FALSE;
			收集工位放收集瓶完成:=FALSE;
			FunctionID:=12;
			ParameterList8:=4;                               //到收集工位取收集瓶
			Execute:=1;
			取收集瓶放暂存工位step:=6;
		END_IF
	6:
		
		IF  RO_ParameterList8=4 AND Status=2 THEN
			取收集瓶放暂存工位step:=10;
			收集工位机器人放收集瓶到暂存工位完成:=TRUE;
			Execute:=0;
		END_IF
	10:
		IF Status=0 THEN
			ParameterList8:=5;                               //放收集瓶到暂存工位
			Execute:=1;
			ParameterList9:=collect_Consume_Slot;
			取收集瓶放暂存工位step:=20;
		END_IF
	20:
		IF RO_ParameterList8=5 AND Status=2 THEN                         //放收集瓶到暂存工位完成
			Execute:=0;
			取收集瓶放暂存工位step:=0;
			取收集瓶放暂存工位完成:=TRUE;
		END_IF
END_CASE
END_ACTION

ACTION A10_取升降机硅胶板:


CASE 取升降硅胶板step OF
		0:
			地轨轴11YDATE.fAbsTarget:=HMI_地轨轴11Y.position[1];     //地轨去上样点样位置
			地轨轴11YDATE.xMoveAbs:=TRUE;
			IF 地轨轴11YDATE.bAbMoveDone THEN
				地轨轴11YDATE.xMoveAbs:=FALSE; 
				IF 升降上料伺服允许取料 AND Status=0 THEN
					FunctionID:=1;                              //取升降硅胶板ID
					ParameterList4:=1;                           //去升降机构位置
					Execute:=1;                                  //机器人启动 
					取升降硅胶板step:=10;
				END_IF
			END_IF
			
		10:
			IF RO_ParameterList4=1 THEN                   //机器人到位
				升降上料机器人已吸住物料:=TRUE;
				取升降硅胶板step:=15;
			END_IF
		15:
			IF 升降上料伺服下降完成  THEN
				ParameterList4:=2;                        //机器人取物料
				取升降硅胶板step:=20;
			END_IF
			
		20:
			IF RO_ParameterList4=2 AND Status=2 THEN                //机器人取物料完成
				ParameterList4:=0;
				Execute:=0;
				升降上料机器人取料完成:=TRUE;
				取升降硅胶板完成:=TRUE;
				取升降硅胶板step:=0;
			END_IF
END_CASE
END_ACTION

ACTION A70_取暂存收集器组放仓库:


CASE 取暂存收集器组放仓库step OF
	0:
		IF RO_ParameterList3=2 THEN
			Execute:=0; 
			地轨轴11YDATE.fAbsTarget:=HMI_地轨轴11Y.position[3];     //地轨去取收集组位置暂存位置
			地轨轴11YDATE.xMoveAbs:=TRUE;
			取暂存收集器组放仓库step:=10;
			粉末收集器定位自动:=FALSE;
		END_IF
	10:
		IF 地轨轴11YDATE.bAbMoveDone AND  Status=0 THEN
			地轨轴11YDATE.xMoveAbs:=FALSE;
			粉末收集器定位自动:=FALSE;
			溶液收集瓶定位自动:=FALSE;
			FunctionID:=14;                              //放收集器/瓶到仓库
			ParameterList6:=15;                          //取暂存收集器组
			Execute:=1; 
			取暂存收集器组放仓库step:=20;
		END_IF
	20:
		IF RO_ParameterList6=15 AND  Status=2 THEN                      //取完成
			Execute:=0; 
			地轨轴11YDATE.fAbsTarget:=HMI_地轨轴11Y.position[6];     //地轨去放收集组位置
			地轨轴11YDATE.xMoveAbs:=TRUE;
			取暂存收集器组放仓库step:=30;
		END_IF
	30:
		IF 地轨轴11YDATE.bAbMoveDone AND  Status=0 THEN
			地轨轴11YDATE.xMoveAbs:=FALSE;
			ParameterList6:=scrape_Old_Plate_Slot;               //取暂存收集器组
			Execute:=1;
			取暂存收集器组放仓库step:=40;
		END_IF
	40:
		IF RO_ParameterList6=scrape_Old_Plate_Slot AND Status=2 THEN
			Execute:=0;
			取暂存收集器组放仓库完成:=TRUE;
			取暂存收集器组放仓库step:=0;
		END_IF
	
END_CASE
END_ACTION

ACTION A32_取拍照硅胶板:
CASE 取拍照硅胶完step OF
	0:
		地轨轴11YDATE.fAbsTarget:=HMI_地轨轴11Y.position[2];     //地轨去刮板拍照位
		地轨轴11YDATE.xMoveAbs:=TRUE;
		IF 地轨轴11YDATE.bAbMoveDone THEN
				地轨轴11YDATE.xMoveAbs:=FALSE;
				取拍照硅胶完step:=5;
		END_IF
	5:		
		IF (拍照工位允许取硅胶板去展开 OR 拍照工位允许取硅胶板放废料区) AND Status=0 THEN    
			FunctionID:=6;                              
			ParameterList5:=6;                           //机器人取硅胶板
			Execute:=1;             
			拍照工位允许取硅胶板去展开 := FALSE;
			取拍照硅胶完step:=10;
		END_IF
	10:
		IF RO_ParameterList5=6 AND Status=2 THEN
			Execute:=0;
			ParameterList6:=0;
			取拍照硅胶板完成:=TRUE;
			取拍照硅胶完step:=0;
		IF 拍照工位允许取硅胶板放废料区 THEN
			拍照工位机器人取硅胶板完成 := TRUE;
		END_IF
		END_IF
END_CASE
END_ACTION

END_PROGRAM

// Device/Application/25_FB_功能块/FB_RB_Control
FUNCTION_BLOCK FB_RB_Control
VAR_INPUT
	StartCmd     : BOOL;
StopCmd      : BOOL;
PauseCmd     : BOOL;
Reset:BOOL;
RobotRunning : BOOL;
RobotStopped : BOOL;
RobotPaused  : BOOL;
RobotAlarm   : BOOL;
PowerOn:BOOL;
END_VAR
VAR_OUTPUT
	StartOut     : BOOL;
StopOut      : BOOL;
PauseOut     : BOOL;
ResetOut:BOOL;
StatusRun    : BOOL;
StatusStop   : BOOL;
StatusPause  : BOOL;
StatusAlarm  : BOOL;
PowerOnOut:BOOL;
END_VAR
VAR
	State        : INT := 0;   // 当前状态
END_VAR

(* ================= 报警优先 ================= *)
IF RobotAlarm THEN
    State := 4;
END_IF

CASE State OF

    (* -------- 0：空闲 -------- *)
    0:
        StartOut := FALSE;
        StopOut  := TRUE;
        PauseOut := FALSE;
		ResetOut:=FALSE;
        IF StartCmd AND NOT RobotAlarm THEN
            State := 1;
        END_IF

    (* -------- 1：运行 -------- *)
    1:
		IF NOT PowerOn THEN
			PowerOnOut:=TRUE;
		ELSE
			PowerOnOut:=FALSE;
		END_IF
		IF PowerOn THEN
			StartOut := TRUE;
			StopOut  := FALSE;
			PauseOut := FALSE;
		END_IF
        

        IF StopCmd THEN
            State := 3;
        ELSIF PauseCmd THEN
            State := 2;
        
        END_IF

    (* -------- 2：暂停 -------- *)
    2:
        PauseOut := TRUE;
		StartOut := FALSE ;
        StopOut  := FALSE;
        IF StopCmd THEN
            State := 3;
        ELSIF  StartCmd AND NOT RobotAlarm THEN
            State := 1;
        END_IF

    (* -------- 3：停止 -------- *)
    3:
        StartOut := FALSE;
        StopOut  := TRUE;
        PauseOut := FALSE;

        IF RobotStopped THEN
            State := 0;
        END_IF

    (* -------- 4：报警 -------- *)
    4:
        StartOut := FALSE;
        StopOut  := TRUE;
        PauseOut := FALSE;

        IF  Reset THEN
			ResetOut:=TRUE;
            State := 0;
        END_IF

END_CASE

(* ================= 状态输出 ================= *)
StatusRun   := (State = 1);
StatusPause := (State = 2);
StatusStop  := (State = 0) OR (State = 3);
StatusAlarm := (State = 4);

END_FUNCTION_BLOCK

// Device/Application/40_Man/Sample_point_sampling_上样点样
PROGRAM Sample_point_sampling_上样点样
VAR
	初始化step: INT;
	清洗step: INT;
	清洗计数: INT;
	上样准备step: INT;
	放硅胶板STEP: INT;
	吸收液体step: INT;
	TON_0: TON;
	TON_1: TON;
	点样step: INT;
	stepTimer           : TON;       // 步骤内通用定时器（调试期模拟，实机替换为FB完成信号）
    bubbleIndex         : INT;       // Step 20 气泡序列循环索引
    cleanCounter        : INT;       // Step 10 清洗循环计数器
	泵初始化完成: BOOL;
	R_TRIG: ARRAY[1..12] OF R_TRIG;
	N: INT;
	A: INT;
	TON: ARRAY[1..11] OF TON;
	打样伺服移动step: INT;
	
	L2_StartTrig : R_TRIG;            // Sampling_L2_Start 上升沿检测器
END_VAR

IF (Sampling_ControlMode = 1) AND (Sampling_L2_State = 10) THEN
	IF (NOT 急停) OR (MODE_State <> 1) THEN
		Sampling_L2_ErrorCode    := 401;       // 急停或模式切换中断
		Sampling_L2_SafeState    := 90;        // RECOVERY_REQUIRED
		Sampling_L2_Retryable    := FALSE;
		Sampling_L2_CompletedSeq := Sampling_L2_AcceptedSeq;
		Sampling_L2_State        := 50;        // INTERRUPTED
	END_IF
END_IF

IF Sampling_X_coordinate>0 THEN 
TON[11](IN:=NOT 上样料架检测1 OR NOT 上样料架检测2,PT:=T#3S);
	IF TON[11].Q THEN
		上样料架报警:=TRUE;
	END_IF
END_IF

// ── 1. 急停联锁（最高优先级）──
IF NOT 急停 THEN
    Sampling_Step  := 0;
    Sampling_Done  := FALSE;
    Sampling_Error := TRUE;
    Sampling_Busy  := FALSE;
	初始化step:=0;
	清洗step:=0;
	清洗计数:=0;
	上样准备step:=0;
	放硅胶板STEP:=0;
	吸收液体step:=0;
	打样伺服移动step:=0;
	泵初始化完成:=FALSE;
	N:=0;
	A:=0;
    stepTimer(IN := FALSE, PT := T#0S);
    RETURN;
END_IF

// ── 2. 复位脉冲（用于错误恢复 / 强制清状态）──
IF Sampling_Reset THEN
    Sampling_Step  := 0;
    Sampling_Done  := FALSE;
    Sampling_Error := FALSE;
    Sampling_Busy  := FALSE;
    stepTimer(IN := FALSE, PT := T#0S);
    cleanCounter := 0;
    bubbleIndex  := 0;
    RETURN;
END_IF

// ── 3. Enable=FALSE 时清 Done（次周期复位握手）──
IF NOT Sampling_Enable THEN
    Sampling_Done := FALSE;
END_IF

// ── 4. 派生 Sampling_Busy（写者唯一：本 POU 是唯一写者，禁止他处赋值）──
Sampling_Busy := (Sampling_Step >= 10)
              AND (Sampling_Step <= 80)
              AND (NOT Sampling_Done);

IF MODE_State=1 THEN
	IF Sampling_ControlMode = 0 THEN     // LEGACY (默认, 行为与今天完全一致)
		CASE Sampling_Step OF
			0:  // ═══ 空闲：等待 Enable 上升 ═══
				IF Sampling_Enable AND (NOT Sampling_Done) THEN
					Sampling_Step := 5;
					stepTimer(IN := FALSE, PT := T#0S);  // 复位定时器
				END_IF
			5:
					A00_initialization_初始化();
					IF Sampling_initialization_OK THEN
						Sampling_initialization_OK:=FALSE;
						Sampling_Step:=10;
					END_IF
			10: // ═══ 清洗（消费 Sampling_clean_instructions + Sampling_clean_count）═══
				A10_clean_清洗();
				IF Sampling_Cleaning_OK THEN
					stepTimer(IN := FALSE, PT := T#0S);
					Sampling_Cleaning_OK:=FALSE;
					Sampling_Step := 20;
				END_IF
	
			20: // ═══ 上样准备 ═══
					A30_Sample_preparation_上样准备();
					IF Sampling_preparation_OK THEN
						Sampling_preparation_OK:=FALSE;
						Sampling_Step:=30;
					END_IF
			 30: // ═══ 放硅胶板（机械臂+传感器自治）═══
				A20_Place_materials_放硅胶板();
				IF Sampling_Place_materials_OK THEN
					Sampling_Place_materials_OK:=FALSE;
					stepTimer(IN := FALSE, PT := T#0S);
					Sampling_Step := 40;
				END_IF	
	
			40: // ═══ 吸液（消费 Sampling_X/Y_coordinate + Sampling_aspirate_instructions）═══
				A40_absorb_liquid_吸收液体();
				IF Sampling_liquid_absorption THEN
					Sampling_liquid_absorption:=FALSE;
					stepTimer(IN := FALSE, PT := T#0S);
					Sampling_Step := 50;
				END_IF
			50: // ═══ 点样（消费 Sampling_dispense_instructions）═══
				A50_Spray_sample_点样();
				IF Sampling_Spray_sample_OK  THEN
					Sampling_Spray_sample_OK:=FALSE;
					Sampling_Step := 60;
					
				END_IF
			60:
				IF  取点样硅胶板完成 THEN
					取点样硅胶板完成:=FALSE;
					stepTimer(IN := FALSE, PT := T#0S);
					Sampling_Done := TRUE;
					Sampling_Busy := FALSE;
					Sampling_Step := 0;
				END_IF
		
			90: // ═══ 故障态：等待外部 Sampling_Reset 脉冲 ═══
				Sampling_Error := TRUE;   // 故障态本身不动作，仅等待顶部复位逻辑
		END_CASE	
	ELSE                                  // L2
		Sampling_L2_Dispatch();
	END_IF
END_IF

ACTION A20_Place_materials_放硅胶板:



	CASE 放硅胶板STEP OF
	 	0:
			点样轴7YDATE.fAbsTarget:=HMI_点样轴7Y.position[1];
			点样轴7YDATE.xMoveAbs:=TRUE;
			放硅胶板STEP:=10;
		10:
			IF 点样轴7YDATE.bAbMoveDone THEN
				上样点样允许放硅胶板:=TRUE;
				点样轴7YDATE.xMoveAbs:=FALSE;
				放硅胶板STEP:=20;
			END_IF
		20:
			IF 上样点样放硅胶板完成 THEN
				上样点样允许放硅胶板:=FALSE;
				上样点样放硅胶板完成:=FALSE;
				上样定位自动:=TRUE;
				Sampling_Place_materials_OK:=TRUE;
				放硅胶板STEP:=0;
			END_IF
		
		
	 END_CASE
END_ACTION

ACTION A30_Sample_preparation_上样准备:
TON[2](IN:=上样准备step=2,PT:=T#0.5S);
R_TRIG[3](CLK:=%MX2005.5 , Q=> );  //泵空闲中

CASE 上样准备step OF
	0:
		上样轴5Z轴DATE.fAbsTarget:=0;
		上样轴5Z轴DATE.xMoveAbs:=TRUE;
		IF 上样轴5Z轴DATE.bAbMoveDone THEN
			N:=1;
			上样轴5Z轴DATE.xMoveAbs:=FALSE ;
			上样准备step:=1;
		END_IF
		
	1:
	
		CASE N OF
			1,2:
				IF %MW1300=0 AND NOT 泵站位符 THEN
					泵站位符:=TRUE;
					转发转存:=Sampling_prep_instructions[N];    
					%MW1300:=LEN(STR:= 转发转存);   //发送字节数
					上样准备step:=2;
				END_IF
		END_CASE
		
	2:
		IF %MW1300=0 AND TON[2].Q THEN 
		转发转存:='/4Q$R';          //查询泵状态指令
		%MW1300:=LEN(STR:= 转发转存);
		END_IF
		
		IF R_TRIG[3].Q THEN
			泵站位符:=FALSE;
			N:=N+1;
			IF N>2 THEN
				
				Sampling_preparation_OK:=TRUE;
				N:=0;
				上样准备step:=0;
			ELSE
				上样准备step:=1;
			END_IF
			
		END_IF
END_CASE
END_ACTION

ACTION A00_initialization_初始化:





CASE 初始化step OF
	0 :
		上样定位手动:=FALSE;
		上样定位自动:=FALSE;
		上样点样三通电池阀手动:=FALSE;
		上样点样三通电池阀自动:=FALSE;
		上样吹气手动:=FALSE;
		上样吹气自动:=FALSE;
		打样瓶上料轴3YDATE.fAbsTarget:=0;
		点样轴6XDATE.fAbsTarget:=0;
		点样轴7YDATE.fAbsTarget:=0;
		上样轴4X轴DATE.fAbsTarget:=0;
		上样轴5Z轴DATE.fAbsTarget:=0;
		上样点样允许放硅胶板:=FALSE;
		点样轴7YDATE.xMoveAbs:=FALSE;
		点样轴6XDATE.xMoveAbs:=FALSE;
		上样轴5Z轴DATE.xMoveAbs:=FALSE;
		上样轴4X轴DATE.xMoveAbs:=FALSE;
		打样瓶上料轴3YDATE.xMoveAbs:=FALSE;
		Sampling_Spray_sample_OK:=FALSE;
		Sampling_liquid_absorption:=FALSE;
		Sampling_preparation_OK:=FALSE;
		上样点样允许取硅胶板:=FALSE;
		上样点样放硅胶板完成:=FALSE;
		大真空泵站位[11]:=FALSE;
		清洗计数:=0;
		清洗step:=0;
		放硅胶板STEP:=0;
		上样准备step:=0;
		吸收液体step:=0;
		点样step:=0;
		初始化step:=5;
	5:
		上样轴5Z轴DATE.fAbsTarget:=0;
		上样轴5Z轴DATE.xMoveAbs:=TRUE;
		IF 上样轴5Z轴DATE.bAbMoveDone THEN
			点样轴7YDATE.fAbsTarget:=0  ;  
			点样轴6XDATE.fAbsTarget:=0  ; 
			上样轴4X轴DATE.fAbsTarget:=0;          
			上样轴4X轴DATE.xMoveAbs:=TRUE;
			点样轴7YDATE.xMoveAbs:=TRUE;
			点样轴6XDATE.xMoveAbs:=TRUE;
			初始化step:=6;
		END_IF
	6:
		IF 上样轴4X轴DATE.bAbMoveDone AND 上样轴5Z轴DATE.bAbMoveDone AND 点样轴6XDATE.bAbMoveDone AND 点样轴7YDATE.bAbMoveDone THEN
			初始化step:=10;
			上样轴4X轴DATE.xMoveAbs:=FALSE;
			点样轴7YDATE.xMoveAbs:=FALSE;
			上样轴5Z轴DATE.xMoveAbs:=FALSE;
			点样轴6XDATE.xMoveAbs:=FALSE;
		END_IF
	10:
		IF %MW1300=0 AND NOT 泵站位符 THEN
			泵站位符:=TRUE;
			转发转存:='/4Z0,1,1R$R';     //泵初始化指令 
			%MW1300:=LEN(STR:= 转发转存);   //发送字节数
			初始化STEP:=20;
		END_IF
	20:
		IF %MW1300=0 THEN
			转发转存:='/4Q$R';          //查询泵状态指令
			%MW1300:=LEN(STR:= 转发转存);
		END_IF
		R_TRIG[1](CLK:=%MX2005.5 , Q=> );  //泵空闲中
		IF R_TRIG[1].Q THEN
			泵站位符:=FALSE;
			初始化STEP:=30;
		END_IF
	30:
		
		
			Sampling_initialization_OK:=TRUE;
			初始化step:=0;
		

END_CASE
END_ACTION

ACTION A50_Spray_sample_点样:
TON[4](IN:=点样step=20,PT:=T#0.5S);
TON[5](IN:=点样气泡传感器,PT:=T#5S);
TON[7](IN:=点样step=10,PT:=T#0.5S);
R_TRIG[10](CLK:=%MX2005.5 , Q=> );  //泵空闲中

CASE 点样step OF
	0:
		点样轴6XDATE.xMoveAbs:=FALSE;
		点样轴7YDATE.xMoveAbs:=FALSE;
		点样step:=1;
	1:
		点样轴6XDATE.fAbsTarget:=HMI_点样轴6X.position[2];        //起始位
		点样轴7YDATE.fAbsTarget:=HMI_点样轴7Y.position[2];         //起始位
		点样轴6XDATE.xMoveAbs:=TRUE;
		点样轴7YDATE.xMoveAbs:=TRUE;
		点样step:=5;
	5:
		IF 点样轴6XDATE.bAbMoveDone AND 点样轴7YDATE.bAbMoveDone THEN
			点样轴6XDATE.xMoveAbs:=FALSE;
			点样轴7YDATE.xMoveAbs:=FALSE;
			IF  %MW1300=0 AND NOT 泵站位符 THEN
				
				泵站位符:=TRUE;
				转发转存:=Sampling_dispense_instructions[1];
				%MW1300:=LEN(STR:= 转发转存);
				上样点样三通电池阀自动:=TRUE;
				点样step:=10;
			END_IF
		END_IF
	10:
		IF  %MW1300=0 AND TON[7].Q THEN                        
				转发转存:='/4Q$R';          //查询泵状态指令
				%MW1300:=LEN(STR:= 转发转存);
				
				IF R_TRIG[10].Q THEN
					泵站位符:=FALSE;
					
					点样step:=15;
				END_IF
		END_IF
	15:
		IF  %MW1300=0 AND NOT 泵站位符 THEN
			上样吹气自动:=TRUE;
			泵站位符:=TRUE;
			转发转存:=Sampling_dispense_instructions[2];
			%MW1300:=LEN(STR:= 转发转存);
			点样轴6XDATE.fAbsTarget:=HMI_点样轴6X.position[3];             //终点位
			点样轴6XDATE.xMoveAbs:=TRUE;
			点样step:=20;
		END_IF

	20:
		IF  %MW1300=0 AND TON[4].Q THEN                        
				转发转存:='/4Q$R';          //查询泵状态指令
				%MW1300:=LEN(STR:= 转发转存);
				
				IF R_TRIG[10].Q THEN
					泵站位符:=FALSE;
					上样点样三通电池阀自动:=FALSE;
					上样吹气自动:=FALSE;
				END_IF
		END_IF
		CASE 打样伺服移动step OF
			0:
				IF 点样轴6XDATE.bAbMoveDone THEN
					点样轴6XDATE.xMoveAbs:=FALSE;
					IF 泵站位符 THEN
						打样伺服移动step:=10;
					ELSE
						点样step:=30;
					END_IF
					
				END_IF
			10:
				点样轴6XDATE.fAbsTarget:=HMI_点样轴6X.position[2];        //起始位
				点样轴6XDATE.xMoveAbs:=TRUE;
				打样伺服移动step:=20;
			20:
				IF 点样轴6XDATE.bAbMoveDone THEN
					点样轴6XDATE.xMoveAbs:=FALSE;
					打样伺服移动step:=30;
				END_IF
			30:
				点样轴6XDATE.fAbsTarget:=HMI_点样轴6X.position[3];             //终点位
				点样轴6XDATE.xMoveAbs:=TRUE;
				打样伺服移动step:=0;
				
		END_CASE
		
	30:
		点样轴6XDATE.fAbsTarget:=HMI_点样轴6X.position[1];        //清洗位
		点样轴6XDATE.xMoveAbs:=TRUE;
		IF 点样轴6XDATE.bAbMoveDone THEN
			点样轴7YDATE.fAbsTarget:=HMI_点样轴7Y.position[1]; 
			点样轴7YDATE.xMoveAbs:=TRUE;
		
		点样step:=40;
		END_IF
		
	40:
		IF 点样轴7YDATE.bAbMoveDone  THEN
			点样轴6XDATE.xMoveAbs:=FALSE;
			点样轴7YDATE.xMoveAbs:=FALSE;
			上样定位自动:=FALSE;
			上样点样允许取硅胶板:=TRUE;
			Sampling_Spray_sample_OK:=TRUE;
			点样step:=0;
		END_IF
 END_CASE
END_ACTION

ACTION A40_absorb_liquid_吸收液体:
TON_0(IN:=吸收液体step=30, PT:=T#0.5S , Q=> , ET=> );
TON_1(IN:=NOT 点样气泡传感器, PT:=T#5S , Q=> , ET=> );
R_TRIG[10](CLK:=%MX2005.5 , Q=> );  //泵空闲中

IF Sampling_X_coordinate>0 AND  Sampling_Y_coordinate>0  THEN
	CASE 吸收液体step OF
		0:
			上样轴5Z轴DATE.fAbsTarget:=0;
			上样轴5Z轴DATE.xMoveAbs:=TRUE;
			IF 上样轴5Z轴DATE.bAbMoveDone THEN
				上样轴5Z轴DATE.xMoveAbs:=FALSE;
				上样轴4X轴DATE.fAbsTarget:=HMI_上样轴4X轴.position[Sampling_X_coordinate];
				打样瓶上料轴3YDATE.fAbsTarget:=HMI_打样瓶上料轴3Y.position[Sampling_Y_coordinate];
				上样轴4X轴DATE.xMoveAbs:=TRUE;
				打样瓶上料轴3YDATE.xMoveAbs:=TRUE;
				吸收液体step:=10;
			END_IF
		10:
			IF 上样轴4X轴DATE.bAbMoveDone AND 打样瓶上料轴3YDATE.bAbMoveDone THEN
				上样轴4X轴DATE.xMoveAbs:=FALSE;
				打样瓶上料轴3YDATE.xMoveAbs:=FALSE;
				上样轴5Z轴DATE.fAbsTarget:=HMI_上样轴5Z轴.position[2];
				上样轴5Z轴DATE.xMoveAbs:=TRUE;
				吸收液体step:=20;
			END_IF
		20:
			IF 上样轴5Z轴DATE.bAbMoveDone THEN
				上样轴5Z轴DATE.xMoveAbs:=FALSE;
				A:=1;
				吸收液体step:=25;
			END_IF
		25:
			CASE A OF
				1,2:
					IF  %MW1300=0 AND NOT 泵站位符 THEN
						转发转存:=Sampling_sample_instructions[A];   //吸收液体
						%MW1300:=LEN(STR:= 转发转存);
						泵站位符:=TRUE;
						吸收液体step:=30;
					END_IF
			END_CASE
					
		
		30:
			IF  %MW1300=0 AND TON_0.Q THEN                        
				转发转存:='/4Q$R';          //查询泵状态指令
				%MW1300:=LEN(STR:= 转发转存);
				
				IF R_TRIG[10].Q THEN
					泵站位符:=FALSE;
					A:=A+1;
					IF A>2 THEN
						A:=0;
						大真空泵站位[11]:=FALSE;
						吸收液体step:=40;
					ELSE
						吸收液体step:=25;
					END_IF
				END_IF
			END_IF

		40:
			上样轴5Z轴DATE.fAbsTarget:=0;
			上样轴5Z轴DATE.xMoveAbs:=TRUE;
			IF 上样轴5Z轴DATE.bAbMoveDone THEN
				上样轴5Z轴DATE.xMoveAbs:=FALSE;
				Sampling_liquid_absorption:=TRUE;
				吸收液体step:=0;
			END_IF

	END_CASE
END_IF
END_ACTION

ACTION Sampling_L2_Dispatch:
L2_StartTrig(CLK := Sampling_L2_Start);

CASE Sampling_L2_State OF

	0:  // ═══ IDLE: 等待 Start 上升沿 ═══
		Sampling_L2_Step := 0;
		IF L2_StartTrig.Q THEN
			// 锁存请求 (序号与动作码一并冻结, 防主机中途改写)
			Sampling_L2_AcceptedSeq := Sampling_L2_RequestSeq;
			Sampling_L2_ActiveCode  := Sampling_L2_ActionCode;
			Sampling_L2_ErrorCode   := 0;
			Sampling_L2_Retryable   := FALSE;
			IF (Sampling_L2_ActionCode = 10)
			   OR (Sampling_L2_ActionCode = 20)
			   OR (Sampling_L2_ActionCode = 60)
			   OR (Sampling_L2_ActionCode = 70) THEN
				// 复位所有 A 动作局部步进 (与本 POU 急停复位块同一集合)
				初始化step := 0;
				清洗step := 0;
				清洗计数 := 0;
				上样准备step := 0;
				放硅胶板STEP := 0;
				吸收液体step := 0;
				打样伺服移动step := 0;
				泵初始化完成 := FALSE;
				N := 0;
				A := 0;
				Sampling_L2_SafeState := 0;       // UNKNOWN (运行中)
				Sampling_L2_State := 10;           // RUNNING
			ELSE
				// 未知动作码 -> 接受前拒绝 (可重试)
				Sampling_L2_ErrorCode    := 101;
				Sampling_L2_Retryable    := TRUE;
				Sampling_L2_CompletedSeq := Sampling_L2_AcceptedSeq;
				Sampling_L2_State        := 30;    // REJECTED
			END_IF
		END_IF

	10: // ═══ RUNNING: 按 ActiveCode 调对应 A 动作, 监视其完成标志 ═══
		CASE Sampling_L2_ActiveCode OF
			10:  // 初始化
				A00_initialization_初始化();
				Sampling_L2_Step := 初始化step;
				IF Sampling_initialization_OK THEN
					Sampling_initialization_OK := FALSE;
					Sampling_L2_SafeState    := 10;   // READY
					Sampling_L2_CompletedSeq := Sampling_L2_AcceptedSeq;
					Sampling_L2_State        := 20;   // DONE
				END_IF
			20:  // 清洗
				A10_clean_清洗();
				Sampling_L2_Step := 清洗step;
				IF Sampling_Cleaning_OK THEN
					Sampling_Cleaning_OK := FALSE;
					Sampling_L2_CompletedSeq := Sampling_L2_AcceptedSeq;
					Sampling_L2_State        := 20;   // DONE
				END_IF
			60:  // 吸样
				A40_absorb_liquid_吸收液体();
				Sampling_L2_Step := 吸收液体step;
				IF Sampling_liquid_absorption THEN
					Sampling_liquid_absorption := FALSE;
					Sampling_L2_CompletedSeq := Sampling_L2_AcceptedSeq;
					Sampling_L2_State        := 20;   // DONE
				END_IF
			70:  // 点样
				A50_Spray_sample_点样();
				Sampling_L2_Step := 点样step;
				IF Sampling_Spray_sample_OK THEN
					Sampling_Spray_sample_OK := FALSE;
					Sampling_L2_CompletedSeq := Sampling_L2_AcceptedSeq;
					Sampling_L2_State        := 20;   // DONE
				END_IF
		END_CASE

	20, 30, 40, 50:  // ═══ 终态: 保持到 Start 落沿或 L2_Reset, 再回 IDLE ═══
		IF (NOT Sampling_L2_Start) OR Sampling_L2_Reset THEN
			Sampling_L2_State := 0;
		END_IF

END_CASE
END_ACTION

ACTION A10_clean_清洗:
TON[1](IN:=清洗step=20,PT:=T#0.5S);
TON[6](IN:=清洗step=40,PT:=T#0.5S);
TON[8](IN:=清洗step=26,PT:=T#0.5S);
R_TRIG[2](CLK:=%MX2005.5 , Q=> );  //泵空闲中
R_TRIG[11](CLK:=%MX2005.5 , Q=> );  //泵空闲中
R_TRIG[12](CLK:=%MX2005.5 , Q=> );  //泵空闲中

CASE 清洗step OF
	0 :
		点样轴6XDATE.xMoveAbs:=FALSE;
		上样轴4X轴DATE.xMoveAbs:=FALSE;
		上样轴5Z轴DATE.xMoveAbs:=FALSE;
		清洗step:=5;
	5:
		点样轴6XDATE.fAbsTarget:=HMI_点样轴6X.position[1];               //6X清洗位置赋值
		上样轴4X轴DATE.fAbsTarget:=HMI_上样轴4X轴.position[9];           //4X清洗位置赋值
		点样轴6XDATE.xMoveAbs:=TRUE;
		上样轴4X轴DATE.xMoveAbs:=TRUE;
		清洗计数:=0;
		清洗step:=6;
	6:
		IF 上样轴4X轴DATE.bAbMoveDone THEN
			上样轴4X轴DATE.xMoveAbs:=FALSE;
			上样轴5Z轴DATE.fAbsTarget:=HMI_上样轴5Z轴.position[1];
			上样轴5Z轴DATE.xMoveAbs:=TRUE;
			清洗step:=7;
		END_IF

	7:
		IF  上样轴5Z轴DATE.bAbMoveDone AND 点样轴6XDATE.bAbMoveDone THEN
			上样轴5Z轴DATE.xMoveAbs:=FALSE;
			点样轴6XDATE.xMoveAbs:=FALSE;
			IF Sampling_clean_count>0 THEN
				清洗step:=10;
			ELSE
				清洗step:=60;
			END_IF
			
		END_IF
	10:
		IF %MW1300=0 AND NOT 泵站位符 THEN
			泵站位符:=TRUE;
			转发转存:=Sampling_clean_instructions[1];    
			%MW1300:=LEN(STR:= 转发转存);   //发送字节数
			大真空泵站位[11]:=TRUE;
			上样点样三通电池阀自动:=TRUE;
			清洗step:=20;
		END_IF
	20:
		IF %MW1300=0 AND TON[1].Q THEN
		转发转存:='/4Q$R';          //查询泵状态指令
		%MW1300:=LEN(STR:= 转发转存);
		END_IF
		
		IF R_TRIG[2].Q THEN
			上样点样三通电池阀自动:=FALSE;
			泵站位符:=FALSE;
			清洗step:=24;
		END_IF
	24:
		IF %MW1300=0 AND NOT 泵站位符 THEN
			泵站位符:=TRUE;
			转发转存:=Sampling_clean_instructions[1];    
			%MW1300:=LEN(STR:= 转发转存);   //发送字节数
			清洗step:=26;
		END_IF
	26:
		IF %MW1300=0 AND TON[8].Q THEN
		转发转存:='/4Q$R';          //查询泵状态指令
		%MW1300:=LEN(STR:= 转发转存);
		END_IF
		
		IF R_TRIG[11].Q THEN
			
			泵站位符:=FALSE;
			清洗step:=30;
		END_IF
	30:
		IF %MW1300=0 AND NOT 泵站位符 THEN
			泵站位符:=TRUE;
			转发转存:=Sampling_clean_instructions[2];    
			%MW1300:=LEN(STR:= 转发转存);   //发送字节数
			
			清洗step:=40;
		END_IF
				
	40:
		IF %MW1300=0 AND TON[6].Q THEN
		转发转存:='/4Q$R';          //查询泵状态指令
		%MW1300:=LEN(STR:= 转发转存);
		END_IF
		
		IF R_TRIG[12].Q THEN
			泵站位符:=FALSE;
			清洗step:=50;
		END_IF
	50:
		清洗计数:=清洗计数+1;
		IF  Sampling_clean_count> 清洗计数 THEN                 
			转发转存:='';
			%MW1300:=128;
			清洗step:=10;
		ELSIF  Sampling_clean_count<= 清洗计数 THEN
			转发转存:='';
			%MW1300:=128;
			清洗计数:=0;
			Sampling_Cleaning_OK:=TRUE;
			清洗step:=0;
		END_IF	
		上样点样三通电池阀自动:=FALSE;
		
	60:
		大真空泵站位[11]:=FALSE;
		Sampling_Cleaning_OK:=TRUE;
		清洗step:=0;
END_CASE
END_ACTION

END_PROGRAM

// Device/Application/40_Man/Collection_process_收集流程
PROGRAM Collection_process_收集流程
VAR
	准备step: INT;
	收集step: INT;
	TON_0: TON;
	搬运step: INT;
	ton3s: TON;
	ton5s: TON;
	i: INT;
	stepTimer: TON;
	R_TRIG: ARRAY[1..5] OF R_TRIG;
	泵初始化完成: BOOL;
	初始化STEP: INT;
	ton: ARRAY[1..10] OF TON;
	L2_StartTrig : R_TRIG;            // Collect_L2_Start 上升沿检测器
	L2_SubStep   : INT;              // collect(20) 子序列步进 (0=准备 1=收集 2=搬运)
END_VAR

// TON自复位：Q变TRUE后IN立即变FALSE，下周期复位，形成循环脉冲
// ton3s(IN := bEnable AND NOT ton3s.Q, PT := T#3S);
// 
// Q脉冲时翻转输出（Q仅维持一个周期，无需上升沿检测）
// IF ton3s.Q THEN
//     bOutput := NOT bOutput;
// END_IF

IF (Collect_ControlMode = 1) AND (Collect_L2_State = 10) THEN
	IF (NOT 急停) OR (MODE_State <> 1) THEN
		Collect_L2_ErrorCode    := 401;
		Collect_L2_SafeState    := 90;
		Collect_L2_Retryable    := FALSE;
		Collect_L2_CompletedSeq := Collect_L2_AcceptedSeq;
		Collect_L2_State        := 50;     // INTERRUPTED
	END_IF
END_IF

// ── 1. 急停联锁（最高优先级）──
IF NOT 急停 THEN
    collect_Step  := 0;
    collect_Done  := FALSE;
    collect_Error := TRUE;
    collect_Busy  := FALSE;
	准备step:=0;
	收集step:=0;
	搬运step:=0;
	初始化STEP:=0;
	泵初始化完成:=FALSE;
    stepTimer(IN := FALSE, PT := T#0S);
    RETURN;
END_IF

// ── 2. 复位脉冲（用于错误恢复 / 强制清状态）──
IF collect_Reset THEN
    collect_Step  := 0;
    collect_Done  := FALSE;
    collect_Error := FALSE;
    collect_Busy  := FALSE;
    stepTimer(IN := FALSE, PT := T#0S);
    RETURN;
END_IF

// ── 3. Enable=FALSE 时清 Done（次周期复位握手）──
//    上位机收到 Done 后会拉低 collect_Enable，本段确保下一周期 Done 自动归零，
//    避免 Done 残留导致 step 0 误判。
IF NOT collect_Enable THEN
    collect_Done := FALSE;
END_IF

// ── 4. 派生 collect_Busy（写者唯一：本 POU 是唯一写者，禁止他处赋值）──
collect_Busy := (collect_Step >= 10)
                    AND (collect_Step <= 80)
                    AND (NOT collect_Done);

IF MODE_State=1 THEN
	IF Collect_ControlMode = 0 THEN       // LEGACY (默认)
		CASE collect_Step OF
			0 :                      // 空闲：等待 Enable 上升
				 IF collect_Enable AND (NOT collect_Done) THEN
					collect_Step := 5;
				 END_IF
			
			5:	
				A00_initialization_初始化();
				IF 收集平台下压气缸原点 AND 收集平台夹持气缸原点 AND 收集平台升降气缸原点 AND 收集平台推出气缸原点 AND 泵初始化完成 THEN
					collect_Step:=10;
					泵初始化完成:=FALSE;
				END_IF
				
				
					
			10:                    //就位
					A10_preparation_准备();
				IF collect_prepare_OK THEN
					collect_prepare_OK:=FALSE;
					collect_Step:=20;
				END_IF
				
				
				
			20:                    //收集    	
				A20_collect_收集();
				IF collect_OK THEN
					
					FOR i := 1 TO collect_count BY 1 DO
						;   // 占位：单次打液动作（实机替换为真实调用）
					END_FOR
					collect_OK:=FALSE;
					collect_Step:=30;
				END_IF
				
				
			30:                    //物料搬运
				A30_transport_物料搬运();
				 IF 收集工位放收集器完成 THEN
					 收集工位放收集器完成:=FALSE;
					collect_Done := TRUE;
					collect_Step:=0;
				 END_IF	
				 
				 
			90: // 故障：等待外部 collect_Reset 脉冲（已在顶部统一处理）
				collect_Error := TRUE;   // 故障态本身不动作，仅等待复位
		END_CASE
	ELSE                                   // L2
		Collect_L2_Dispatch();
	END_IF
END_IF

ACTION A20_collect_收集:
ton[1](IN:=收集step=10,PT:=T#0.5S);
ton[2](IN:=收集step=30,PT:=T#10S);
R_TRIG[5](CLK:=%MX2005.5 , Q=> );  //泵空闲中
CASE 收集step OF
	0 :
		IF collect_forward_instructions<>'' THEN
			收集进液自动:=TRUE;
			
			
		END_IF
		IF %MW1300=0 AND 泵站位符=FALSE  THEN
			转发转存:=collect_forward_instructions; 
			%MW1300:=LEN(STR:= 转发转存);   //发送字节数
			泵站位符:=TRUE;
			收集step:=10;
		END_IF
	10:
		IF %MW1300=0 AND ton[1].Q THEN
			转发转存:='/3Q$R';          //查询泵状态指令
			%MW1300:=LEN(STR:= 转发转存);
		END_IF
		
		
		IF R_TRIG[5].Q THEN
			泵站位符:=FALSE;
			收集step:=20;
		END_IF
	

	20:
		IF TRUE  THEN    //注射泵完成//
			转发转存:='';
			%MW300:=128;
			收集进液自动:=FALSE;
			收集排液自动:=TRUE;
			收集正压排液自动:=TRUE;
			收集计数:=收集计数+1;
			收集step:=30;
		END_IF
	30:
		IF ton[2].Q THEN
			TON_0(IN:=TRUE, PT:=T#5S , Q=> , ET=> );
			IF 收集计数>=collect_count AND TON_0.Q THEN
				收集计数:=0;
				收集step:=40;
			ELSE
				收集排液自动:=FALSE;
				收集正压排液自动:=FALSE;
				收集step:=0;
			END_IF
		END_IF
	40:
		
			收集排液自动:=FALSE;
			收集正压排液自动:=FALSE;
			collect_OK:=TRUE;
			收集step:=0;

		

		
END_CASE
END_ACTION

ACTION A00_initialization_初始化:
R_TRIG[1](CLK:=%MX2005.5 , Q=> );  //泵空闲中

//初始化流程
CASE 初始化STEP OF
	0:
		收集下压气缸手动:=FALSE;
		收集下压气缸自动:=FALSE;
		收集夹持气缸手动:=FALSE;
		收集夹持气缸自动:=FALSE;
		收集升降气缸手动:=FALSE;
		收集升降气缸自动:=FALSE;
		收集伸缩气缸手动:=FALSE;
		收集伸缩气缸自动:=FALSE;
		收集进液手动:=FALSE;
		收集进液自动:=FALSE;
		收集排液手动:=FALSE;
		收集排液自动:=FALSE;
		收集正压排液手动:=FALSE;
		收集正压排液自动:=FALSE;
		溶液收集瓶定位手动:=FALSE;
		收集工位允许放收集瓶:=FALSE;
		收集工位允许放收集器:=FALSE;
		收集工位允许机器人退出工位:=FALSE;
		收集工位允许机器人取收集瓶放暂存工位:=FALSE;
		收集工位允许取收集器:=FALSE;
		收集工位机器人取收集器放回暂存工位:=FALSE;
		
	
		收集工位放收集瓶完成:=FALSE;
		收集工位放收集器到工位:=FALSE;
	
		收集工位机器人退出完成:=FALSE;
		
		收集工位机器人放收集瓶到暂存工位完成:=FALSE;
		
		收集工位机器人到达收集器位置:=FALSE;

		collect_prepare_OK:=FALSE;
		collect_OK:=FALSE;
		收集工位放收集器完成:=FALSE;
		收集step:=0;
		准备step:=0;
		搬运step:=0;
		IF %MW1300=0 AND NOT 泵站位符 THEN
			泵站位符:=TRUE;
			转发转存:='/3Z0,2,2R$R';     //泵初始化指令 
			%MW1300:=LEN(STR:= 转发转存);   //发送字节数
			初始化STEP:=10;
		END_IF
	10:
		IF %MW1300=0 THEN
			转发转存:='/3Q$R';          //查询泵状态指令
			%MW1300:=LEN(STR:= 转发转存);
		END_IF
		
		IF R_TRIG[1].Q THEN
			泵站位符:=FALSE;
			泵初始化完成:=TRUE;
			初始化STEP:=0;
		END_IF
END_CASE
END_ACTION

ACTION Collect_L2_Dispatch:
// 功能:
//   收集 L2 统一动作通道派发器。仅在 MODE_State=1 且 Collect_ControlMode=1 时由
//   POU body 调用 (与 legacy CASE collect_Step 互斥, 单写者)。
L2_StartTrig(CLK := Collect_L2_Start);

CASE Collect_L2_State OF

	0:  // ═══ IDLE ═══
		Collect_L2_Step := 0;
		IF L2_StartTrig.Q THEN
			Collect_L2_AcceptedSeq := Collect_L2_RequestSeq;
			Collect_L2_ActiveCode  := Collect_L2_ActionCode;
			Collect_L2_ErrorCode   := 0;
			Collect_L2_Retryable   := FALSE;
			IF (Collect_L2_ActionCode = 10) OR (Collect_L2_ActionCode = 20) THEN
				// 复位 A 动作局部步进与子序列 (镜像本 POU 急停复位集合)
				准备step := 0;
				收集step := 0;
				搬运step := 0;
				初始化STEP := 0;
				泵初始化完成 := FALSE;
				L2_SubStep := 0;
				Collect_L2_SafeState := 0;
				Collect_L2_State := 10;            // RUNNING
			ELSE
				Collect_L2_ErrorCode    := 101;
				Collect_L2_Retryable    := TRUE;
				Collect_L2_CompletedSeq := Collect_L2_AcceptedSeq;
				Collect_L2_State        := 30;     // REJECTED
			END_IF
		END_IF

	10: // ═══ RUNNING ═══
		CASE Collect_L2_ActiveCode OF
			10:  // 初始化 (镜像 legacy step 5: A00 + 四气缸原点 + 泵初始化完成)
				A00_initialization_初始化();
				Collect_L2_Step := 初始化STEP;
				IF 收集平台下压气缸原点 AND 收集平台夹持气缸原点
				   AND 收集平台升降气缸原点 AND 收集平台推出气缸原点
				   AND 泵初始化完成 THEN
					泵初始化完成 := FALSE;
					Collect_L2_SafeState    := 10;   // READY
					Collect_L2_CompletedSeq := Collect_L2_AcceptedSeq;
					Collect_L2_State        := 20;   // DONE
				END_IF
			20:  // 收集 = 准备 -> 收集 -> 搬运 (镜像 legacy step 10->20->30)
				CASE L2_SubStep OF
					0:
						A10_preparation_准备();
						Collect_L2_Step := 准备step;
						IF collect_prepare_OK THEN
							collect_prepare_OK := FALSE;
							L2_SubStep := 1;
						END_IF
					1:
						A20_collect_收集();
						Collect_L2_Step := 100 + 收集step;
						IF collect_OK THEN
							collect_OK := FALSE;
							L2_SubStep := 2;
						END_IF
					2:
						A30_transport_物料搬运();
						Collect_L2_Step := 200 + 搬运step;
						IF 收集工位放收集器完成 THEN
							收集工位放收集器完成 := FALSE;
							Collect_L2_CompletedSeq := Collect_L2_AcceptedSeq;
							Collect_L2_State        := 20;   // DONE
						END_IF
				END_CASE
		END_CASE

	20, 30, 40, 50:  // ═══ 终态 ═══
		IF (NOT Collect_L2_Start) OR Collect_L2_Reset THEN
			Collect_L2_State := 0;
		END_IF

END_CASE
END_ACTION

ACTION A30_transport_物料搬运:


CASE 搬运step OF
	0 :                     //复位气缸
		收集下压气缸自动:=FALSE;
		
		搬运step:=5;
	5:
		IF 收集平台下压气缸原点 THEN
			收集升降气缸自动:=FALSE;
			搬运step:=10;
		END_IF
	10:                    //复位伸缩气缸
		IF 收集平台升降气缸原点 THEN
			收集伸缩气缸自动:=TRUE;
			搬运step:=20;
		END_IF
	20:                    //允许机器人收集瓶
		IF 收集平台推出气缸动点 THEN
			收集工位允许机器人取收集瓶放暂存工位:=TRUE;
			搬运step:=30;
		END_IF
	30:
		IF 收集工位机器人放收集瓶到暂存工位完成 THEN
			收集工位允许机器人取收集瓶放暂存工位:=FALSE;
			收集工位机器人放收集瓶到暂存工位完成:=FALSE;
			收集伸缩气缸自动:=FALSE;
			收集工位允许取收集器:=TRUE;
			搬运step:=40;
		END_IF
	40:
		IF 收集工位机器人到达收集器位置 THEN
				收集工位机器人到达收集器位置:=FALSE;
			收集夹持气缸自动:=FALSE;
			收集工位允许取收集器:=FALSE;
			搬运step:=50;
		END_IF
	50:
		IF 收集平台夹持气缸原点 THEN
			收集工位机器人取收集器放回暂存工位:=TRUE;
			搬运step:=60;
		END_IF
	60:
		 IF 收集工位放收集器完成 THEN
		 	搬运step:=0;
		 END_IF
		
		
		

END_CASE
END_ACTION

ACTION A10_preparation_准备:
//准备工作
CASE 准备step OF	
	0:
		IF 收集平台夹持气缸原点 AND 收集平台下压气缸原点 THEN
		收集工位允许放收集器:=TRUE;
		准备step:=10;
		END_IF
	10:
		IF 收集工位放收集器到工位 THEN
			收集夹持气缸自动:=TRUE;
			收集工位允许放收集器:=FALSE;
			准备step:=20;
		END_IF
	20:
		IF 收集平台夹持气缸动点 THEN
			收集工位允许机器人退出工位:=TRUE;
			准备step:=30;
		END_IF
		
	30:
		IF 收集工位机器人退出完成 THEN
			
